  MoveL 2530 to (-12.23, -53.59, 110) mm, rotated rx 180 ry 0 rz 180 deg; joints [26.087, 43.16, 28.85, -152.762, 73.896, -188.126]
  Call Extruder(23965.750)
  MoveL 2531 to (0, -54.97, 110) mm, rotated rx 180 ry 0 rz -180 deg; joints [25.019, 44.364, 26.268, -153.678, 72.511, -188.456]
  Call Extruder(23973.266)
  MoveL 2532 to (8.41, -54.02, 110) mm, rotated rx -180 ry 0 rz 180 deg; joints [24.593, 45.312, 24.248, -153.968, 71.486, -188.816]
  Call Extruder(23976.680)
  MoveL 2533 to (12.23, -53.59, 110) mm, rotated rx -180 ry 0 rz -180 deg; joints [24.406, 45.751, 23.319, -154.09, 71.016, -188.98]
  Call Extruder(23987.610)
  MoveL 2534 to (23.85, -49.53, 110) mm, rotated rx 180 ry 0 rz 180 deg; joints [24.239, 47.254, 20.153, -154.003, 69.493, -189.695]
  Call Extruder(23998.541)
  MoveL 2535 to (34.27, -42.98, 110) mm, rotated rx -180 ry 0 rz 180 deg; joints [24.487, 48.8, 16.924, -153.451, 68.027, -190.589]
  Call Extruder(24009.471)
  MoveL 2536 to (42.98, -34.27, 110) mm, rotated rx -180 ry 0 rz -180 deg; joints [25.101, 50.315, 13.782, -152.49, 66.697, -191.641]
  Call Extruder(24020.401)
  MoveL 2537 to (49.52, -23.85, 110) mm, rotated rx 180 ry 0 rz 180 deg; joints [26.025, 51.725, 10.877, -151.191, 65.574, -192.812]
  Call Extruder(24031.331)
  MoveL 2538 to (53.59, -12.23, 110) mm, rotated rx 180 ry 0 rz -180 deg; joints [27.2, 52.961, 8.346, -149.634, 64.721, -194.047]
  Call Extruder(24042.261)
  MoveL 2539 to (54.97, 0, 110) mm, rotated rx 180 ry 0 rz 180 deg; joints [28.57, 53.956, 6.315, -147.909, 64.182, -195.275]
  Call Extruder(24053.192)
  MoveL 2540 to (53.59, 12.23, 110) mm, rotated rx 180 ry 0 rz -180 deg; joints [30.077, 54.657, 4.889, -146.106, 63.985, -196.418]
  Call Extruder(24064.122)
  MoveL 2541 to (49.52, 23.85, 110) mm, rotated rx -180 ry 0 rz -180 deg; joints [31.665, 55.023, 4.145, -144.311, 64.137, -197.398]
  Call Extruder(24075.052)
  MoveL 2542 to (42.98, 34.27, 110) mm, rotated rx -180 ry 0 rz -180 deg; joints [33.282, 55.034, 4.123, -142.6, 64.622, -198.143]
  Call Extruder(24085.982)
  MoveL 2543 to (34.27, 42.98, 110) mm, rotated rx 180 ry 0 rz -180 deg; joints [34.874, 54.688, 4.826, -141.036, 65.404, -198.604]
  Call Extruder(24096.912)
  MoveL 2544 to (23.85, 49.53, 110) mm, rotated rx -180 ry 0 rz -180 deg; joints [36.387, 54.006, 6.213, -139.667, 66.431, -198.752]
  Call Extruder(24107.843)
  MoveL 2545 to (12.23, 53.59, 110) mm, rotated rx 180 ry 0 rz 180 deg; joints [37.766, 53.026, 8.211, -138.531, 67.643, -198.581]
  Call Extruder(24118.773)
  MoveL 2546 to (0, 54.97, 110) mm, rotated rx 180 ry 0 rz -180 deg; joints [38.954, 51.803, 10.716, -137.657, 68.971, -198.108]
  Call Extruder(24129.703)
  MoveL 2547 to (-12.23, 53.59, 110) mm, rotated rx 180 ry 0 rz 180 deg; joints [39.895, 50.401, 13.604, -137.075, 70.35, -197.367]
  Call Extruder(24140.633)
  MoveL 2548 to (-23.85, 49.52, 110) mm, rotated rx 180 ry 0 rz 180 deg; joints [40.528, 48.89, 16.735, -136.814, 71.718, -196.406]
  Call Extruder(24151.563)
  MoveL 2549 to (-34.27, 42.98, 110) mm, rotated rx 180 ry 0 rz 180 deg; joints [40.799, 47.344, 19.964, -136.906, 73.02, -195.282]
  Call Extruder(24162.494)
  MoveL 2550 to (-42.98, 34.27, 110) mm, rotated rx 180 ry 0 rz 180 deg; joints [40.659, 45.837, 23.137, -137.381, 74.206, -194.06]
  Call Extruder(24173.424)
  MoveL 2551 to (-49.53, 23.85, 110) mm, rotated rx 180 ry 0 rz 180 deg; joints [40.072, 44.441, 26.103, -138.261, 75.233, -192.812]
  Call Extruder(24184.354)
  MoveL 2552 to (-53.59, 12.23, 110) mm, rotated rx 180 ry 0 rz 180 deg; joints [39.031, 43.225, 28.711, -139.546, 76.062, -191.607]
  Call Extruder(24195.284)
  MoveL 2553 to (-54.97, 0, 110) mm, rotated rx 180 ry 0 rz -180 deg; joints [37.56, 42.249, 30.821, -141.207, 76.654, -190.512]
  Call Extruder(24200.810)
  MoveL 2554 to (-54.27, -6.18, 110) mm, rotated rx 180 ry 0 rz 180 deg; joints [36.644, 41.897, 31.587, -142.193, 76.815, -190.036]
  Set speed (130.0 mm/s)
  MoveL 2555 to (-49.9, -9.51, 110) mm, rotated rx 180 ry 0 rz -180 deg; joints [35.741, 42.07, 31.21, -143.077, 76.496, -189.952]
  MoveL 2556 to (2.97, -12.99, 110) mm, rotated rx 180 ry 0 rz 180 deg; joints [30.614, 47.041, 20.6, -147.387, 70.89, -191.831]
  Call Extruder(24205.473)
  Set speed (80.0 mm/s)
  MoveL 2557 to (5.78, -12.01, 110) mm, rotated rx 180 ry 0 rz 180 deg; joints [30.526, 47.405, 19.836, -147.403, 70.534, -192.029]
  Call Extruder(24210.137)
  MoveL 2558 to (8.31, -10.42, 110) mm, rotated rx 180 ry 0 rz 180 deg; joints [30.538, 47.78, 19.051, -147.312, 70.192, -192.268]
  Call Extruder(24214.801)
  MoveL 2559 to (10.42, -8.31, 110) mm, rotated rx 180 ry 0 rz 180 deg; joints [30.649, 48.146, 18.287, -147.118, 69.881, -192.537]
  Call Extruder(24219.465)
  MoveL 2560 to (12.01, -5.78, 110) mm, rotated rx 180 ry 0 rz 180 deg; joints [30.85, 48.485, 17.579, -146.835, 69.616, -192.823]
  Call Extruder(24224.128)
  MoveL 2561 to (12.99, -2.97, 110) mm, rotated rx 180 ry 0 rz -180 deg; joints [31.131, 48.78, 16.965, -146.478, 69.412, -193.113]
  Call Extruder(24228.792)
  MoveL 2562 to (13.33, 0, 110) mm, rotated rx -180 ry 0 rz -180 deg; joints [31.476, 49.016, 16.474, -146.065, 69.279, -193.391]
  Call Extruder(24233.456)
  MoveL 2563 to (12.99, 2.97, 110) mm, rotated rx 180 ry 0 rz 180 deg; joints [31.869, 49.181, 16.131, -145.619, 69.224, -193.643]
  Call Extruder(24238.120)
  MoveL 2564 to (12.01, 5.78, 110) mm, rotated rx 180 ry 0 rz -180 deg; joints [32.292, 49.267, 15.952, -145.159, 69.248, -193.854]
  Call Extruder(24242.783)
  MoveL 2565 to (10.42, 8.31, 110) mm, rotated rx -180 ry 0 rz 180 deg; joints [32.725, 49.27, 15.947, -144.709, 69.35, -194.015]
  Call Extruder(24247.448)
  MoveL 2566 to (8.31, 10.42, 110) mm, rotated rx -180 ry 0 rz -180 deg; joints [33.149, 49.188, 16.116, -144.289, 69.524, -194.115]
  Call Extruder(24252.111)
  MoveL 2567 to (5.78, 12.01, 110) mm, rotated rx -180 ry 0 rz -180 deg; joints [33.544, 49.027, 16.45, -143.918, 69.761, -194.149]
  Call Extruder(24256.775)
  MoveL 2568 to (2.97, 13, 110) mm, rotated rx -180 ry 0 rz -180 deg; joints [33.893, 48.795, 16.933, -143.612, 70.049, -194.115]
  Call Extruder(24261.439)
  MoveL 2569 to (0, 13.33, 110) mm, rotated rx -180 ry 0 rz 180 deg; joints [34.177, 48.503, 17.54, -143.386, 70.372, -194.014]
  Call Extruder(24266.103)
  MoveL 2570 to (-2.97, 13, 110) mm, rotated rx 180 ry 0 rz 180 deg; joints [34.384, 48.167, 18.243, -143.251, 70.715, -193.854]
  Call Extruder(24270.766)
  MoveL 2571 to (-5.78, 12.01, 110) mm, rotated rx 180 ry 0 rz 180 deg; joints [34.5, 47.802, 19.005, -143.214, 71.061, -193.641]
  Call Extruder(24275.430)
  MoveL 2572 to (-8.31, 10.42, 110) mm, rotated rx 180 ry 0 rz -180 deg; joints [34.518, 47.427, 19.79, -143.279, 71.393, -193.388]
  Call Extruder(24280.094)
  MoveL 2573 to (-10.42, 8.31, 110) mm, rotated rx 180 ry 0 rz -180 deg; joints [34.436, 47.061, 20.556, -143.443, 71.696, -193.109]
  Call Extruder(24284.758)
  MoveL 2574 to (-12.01, 5.78, 110) mm, rotated rx 180 ry 0 rz -180 deg; joints [34.254, 46.723, 21.268, -143.702, 71.956, -192.818]
  Call Extruder(24289.421)
  MoveL 2575 to (-12.99, 2.97, 110) mm, rotated rx -180 ry 0 rz -180 deg; joints [33.981, 46.429, 21.887, -144.044, 72.158, -192.53]
  Call Extruder(24294.085)
  MoveL 2576 to (-13.33, 0, 110) mm, rotated rx 180 ry 0 rz -180 deg; joints [33.63, 46.194, 22.383, -144.454, 72.295, -192.26]
  Call Extruder(24298.749)
  MoveL 2577 to (-13, -2.97, 110) mm, rotated rx 180 ry 0 rz 180 deg; joints [33.218, 46.029, 22.731, -144.91, 72.357, -192.02]
  Call Extruder(24303.413)
  MoveL 2578 to (-12.01, -5.78, 110) mm, rotated rx -180 ry 0 rz -180 deg; joints [32.767, 45.943, 22.912, -145.39, 72.343, -191.823]
  Call Extruder(24308.076)
  MoveL 2579 to (-10.42, -8.31, 110) mm, rotated rx -180 ry 0 rz -180 deg; joints [32.302, 45.941, 22.917, -145.868, 72.25, -191.676]
  Call Extruder(24312.741)
  MoveL 2580 to (-8.31, -10.42, 110) mm, rotated rx 180 ry 0 rz 180 deg; joints [31.85, 46.022, 22.746, -146.317, 72.084, -191.586]
  Call Extruder(24317.404)
  MoveL 2581 to (-5.78, -12.01, 110) mm, rotated rx 180 ry 0 rz -180 deg; joints [31.435, 46.182, 22.408, -146.713, 71.853, -191.557]
  Call Extruder(24322.068)
  MoveL 2582 to (-2.97, -12.99, 110) mm, rotated rx 180 ry 0 rz -180 deg; joints [31.079, 46.413, 21.92, -147.034, 71.566, -191.59]
  Call Extruder(24326.732)
  MoveL 2583 to (0, -13.33, 110) mm, rotated rx 180 ry 0 rz 180 deg; joints [30.801, 46.704, 21.307, -147.262, 71.24, -191.682]
  Call Extruder(24331.396)
  MoveL 2584 to (2.97, -12.99, 110) mm, rotated rx 180 ry 0 rz 180 deg; joints [30.614, 47.041, 20.6, -147.387, 70.89, -191.831]
  Set speed (130.0 mm/s)
  MoveL 2585 to (2.97, -12.99, 115) mm, rotated rx 180 ry 0 rz 180 deg; joints [30.614, 46.171, 20.829, -147.266, 70.35, -192.198]
  MoveL 2586 to (-26.25, -4.54, 115) mm, rotated rx 180 ry 0 rz 180 deg; joints [34.172, 43.696, 25.979, -144.096, 73.299, -191.753]
  Call Extruder(24333.628)
  Set speed (60.0 mm/s)
  MoveL 2587 to (-26.09, -5.96, 115) mm, rotated rx 180 ry 0 rz -180 deg; joints [33.969, 43.617, 26.145, -144.319, 73.328, -191.64]
  Call Extruder(24342.993)
  MoveL 2588 to (-24.12, -11.61, 115) mm, rotated rx -180 ry 0 rz 180 deg; joints [33.033, 43.441, 26.513, -145.31, 73.3, -191.25]
  Call Extruder(24352.358)
  MoveL 2589 to (-20.93, -16.69, 115) mm, rotated rx -180 ry 0 rz -180 deg; joints [32.066, 43.436, 26.524, -146.303, 73.118, -190.96]
  Call Extruder(24361.723)
  MoveL 2590 to (-16.69, -20.93, 115) mm, rotated rx 180 ry 0 rz 180 deg; joints [31.126, 43.602, 26.176, -147.237, 72.789, -190.781]
  Call Extruder(24371.088)
  MoveL 2591 to (-11.61, -24.11, 115) mm, rotated rx 180 ry 0 rz -180 deg; joints [30.272, 43.93, 25.489, -148.057, 72.326, -190.719]
  Call Extruder(24380.453)
  MoveL 2592 to (-5.96, -26.09, 115) mm, rotated rx 180 ry 0 rz -180 deg; joints [29.552, 44.403, 24.5, -148.713, 71.753, -190.773]
  Call Extruder(24389.818)
  MoveL 2593 to (0, -26.77, 115) mm, rotated rx 180 ry 0 rz -180 deg; joints [29.003, 44.998, 23.261, -149.17, 71.098, -190.943]
  Call Extruder(24399.183)
  MoveL 2594 to (5.96, -26.09, 115) mm, rotated rx 180 ry 0 rz 180 deg; joints [28.65, 45.685, 21.836, -149.405, 70.395, -191.222]
  Call Extruder(24408.548)
  MoveL 2595 to (11.61, -24.12, 115) mm, rotated rx -180 ry 0 rz -180 deg; joints [28.503, 46.429, 20.297, -149.412, 69.681, -191.599]
  Call Extruder(24417.913)
  MoveL 2596 to (16.69, -20.93, 115) mm, rotated rx 180 ry 0 rz 180 deg; joints [28.559, 47.193, 18.722, -149.196, 68.995, -192.063]
  Call Extruder(24427.278)
  MoveL 2597 to (20.93, -16.69, 115) mm, rotated rx 180 ry 0 rz -180 deg; joints [28.808, 47.939, 17.188, -148.777, 68.374, -192.593]
  Call Extruder(24436.643)
  MoveL 2598 to (24.12, -11.61, 115) mm, rotated rx 180 ry 0 rz 180 deg; joints [29.229, 48.631, 15.771, -148.183, 67.849, -193.167]
  Call Extruder(24446.008)
  MoveL 2599 to (26.09, -5.96, 115) mm, rotated rx 180 ry 0 rz -180 deg; joints [29.796, 49.233, 14.54, -147.448, 67.449, -193.756]
  Call Extruder(24455.373)
  MoveL 2600 to (26.77, 0, 115) mm, rotated rx -180 ry 0 rz 180 deg; joints [30.482, 49.715, 13.556, -146.614, 67.194, -194.33]
  Call Extruder(24464.738)
  MoveL 2601 to (26.09, 5.96, 115) mm, rotated rx 180 ry 0 rz -180 deg; joints [31.252, 50.053, 12.867, -145.722, 67.097, -194.856]
  Call Extruder(24474.103)
  MoveL 2602 to (24.12, 11.61, 115) mm, rotated rx 180 ry 0 rz -180 deg; joints [32.076, 50.229, 12.509, -144.815, 67.162, -195.304]
  Call Extruder(24483.468)
  MoveL 2603 to (20.93, 16.69, 115) mm, rotated rx 180 ry 0 rz -180 deg; joints [32.917, 50.234, 12.499, -143.935, 67.382, -195.647]
  Call Extruder(24492.833)
  MoveL 2604 to (16.69, 20.93, 115) mm, rotated rx 180 ry 0 rz -180 deg; joints [33.742, 50.068, 12.837, -143.118, 67.744, -195.864]
  Call Extruder(24502.198)
  MoveL 2605 to (11.61, 24.12, 115) mm, rotated rx 180 ry 0 rz -180 deg; joints [34.517, 49.739, 13.507, -142.397, 68.228, -195.943]
  Call Extruder(24511.563)
  MoveL 2606 to (5.96, 26.09, 115) mm, rotated rx -180 ry 0 rz -180 deg; joints [35.208, 49.265, 14.475, -141.802, 68.807, -195.879]
  Call Extruder(24520.928)
  MoveL 2607 to (0, 26.77, 115) mm, rotated rx 180 ry 0 rz 180 deg; joints [35.784, 48.669, 15.692, -141.357, 69.451, -195.676]
  Call Extruder(24530.293)
  MoveL 2608 to (-5.96, 26.09, 115) mm, rotated rx 180 ry 0 rz -180 deg; joints [36.214, 47.982, 17.101, -141.082, 70.128, -195.348]
  Call Extruder(24539.658)
  MoveL 2609 to (-11.61, 24.12, 115) mm, rotated rx 180 ry 0 rz -180 deg; joints [36.473, 47.238, 18.63, -140.991, 70.806, -194.913]
  Call Extruder(24549.023)
  MoveL 2610 to (-16.69, 20.93, 115) mm, rotated rx 180 ry 0 rz -180 deg; joints [36.542, 46.474, 20.205, -141.096, 71.454, -194.397]
  Call Extruder(24558.388)
  MoveL 2611 to (-20.93, 16.69, 115) mm, rotated rx 180 ry 0 rz 180 deg; joints [36.407, 45.728, 21.747, -141.398, 72.042, -193.828]
  Call Extruder(24567.753)
  MoveL 2612 to (-24.12, 11.61, 115) mm, rotated rx 180 ry 0 rz -180 deg; joints [36.065, 45.037, 23.182, -141.894, 72.545, -193.238]
  Call Extruder(24577.118)
  MoveL 2613 to (-26.09, 5.96, 115) mm, rotated rx 180 ry 0 rz 180 deg; joints [35.528, 44.435, 24.434, -142.566, 72.939, -192.658]
  Call Extruder(24586.483)
  MoveL 2614 to (-26.77, 0, 115) mm, rotated rx 180 ry 0 rz 180 deg; joints [34.817, 43.954, 25.439, -143.388, 73.205, -192.117]
  Call Extruder(24591.271)
  MoveL 2615 to (-26.42, -3.05, 115) mm, rotated rx 180 ry 0 rz 180 deg; joints [34.385, 43.78, 25.803, -143.863, 73.268, -191.872]
  Set speed (130.0 mm/s)
  MoveL 2616 to (-41.86, -6.29, 115) mm, rotated rx -180 ry 0 rz 180 deg; joints [35.393, 42.068, 29.404, -143.155, 74.986, -190.985]
  Call Extruder(24596.269)
  Set speed (60.0 mm/s)
  MoveL 2617 to (-41.5, -9.47, 115) mm, rotated rx 180 ry 0 rz -180 deg; joints [34.924, 41.89, 29.78, -143.664, 75.057, -190.74]
  Call Extruder(24611.165)
  MoveL 2618 to (-38.36, -18.47, 115) mm, rotated rx 180 ry 0 rz 180 deg; joints [33.373, 41.609, 30.376, -145.291, 75.032, -190.143]
  Call Extruder(24626.061)
  MoveL 2619 to (-33.29, -26.54, 115) mm, rotated rx -180 ry 0 rz 180 deg; joints [31.763, 41.6, 30.393, -146.935, 74.762, -189.709]
  Call Extruder(24640.957)
  MoveL 2620 to (-26.54, -33.29, 115) mm, rotated rx -180 ry 0 rz 180 deg; joints [30.206, 41.866, 29.831, -148.484, 74.252, -189.449]
  Call Extruder(24655.852)
  MoveL 2621 to (-18.47, -38.36, 115) mm, rotated rx 180 ry 0 rz -180 deg; joints [28.808, 42.391, 28.721, -149.834, 73.522, -189.362]
  Call Extruder(24670.748)
  MoveL 2622 to (-9.47, -41.5, 115) mm, rotated rx 180 ry 0 rz 180 deg; joints [27.654, 43.148, 27.128, -150.897, 72.606, -189.448]
  Call Extruder(24685.644)
  MoveL 2623 to (0, -42.57, 115) mm, rotated rx 180 ry 0 rz -180 deg; joints [26.805, 44.097, 25.141, -151.616, 71.554, -189.702]
  Call Extruder(24697.356)
  MoveL 2624 to (7.45, -41.73, 115) mm, rotated rx 180 ry 0 rz 180 deg; joints [26.398, 44.954, 23.354, -151.89, 70.665, -190.03]
  Call Extruder(24700.540)
  MoveL 2625 to (9.47, -41.5, 115) mm, rotated rx 180 ry 0 rz 180 deg; joints [26.29, 45.19, 22.863, -151.96, 70.422, -190.119]
  Call Extruder(24715.435)
  MoveL 2626 to (18.47, -38.36, 115) mm, rotated rx 180 ry 0 rz -180 deg; joints [26.114, 46.373, 20.412, -151.925, 69.271, -190.691]
  Call Extruder(24730.331)
  MoveL 2627 to (26.54, -33.28, 115) mm, rotated rx 180 ry 0 rz 180 deg; joints [26.262, 47.588, 17.908, -151.532, 68.165, -191.402]
  Call Extruder(24745.227)
  MoveL 2628 to (33.28, -26.54, 115) mm, rotated rx 180 ry 0 rz -180 deg; joints [26.703, 48.777, 15.472, -150.817, 67.162, -192.23]
  Call Extruder(24760.123)
  MoveL 2629 to (38.36, -18.47, 115) mm, rotated rx 180 ry 0 rz 180 deg; joints [27.4, 49.879, 13.221, -149.833, 66.317, -193.141]
  Call Extruder(24775.019)
  MoveL 2630 to (41.51, -9.47, 115) mm, rotated rx 180 ry 0 rz 180 deg; joints [28.309, 50.841, 11.265, -148.64, 65.677, -194.091]
  Call Extruder(24789.914)
  MoveL 2631 to (42.57, 0, 115) mm, rotated rx 180 ry 0 rz 180 deg; joints [29.382, 51.614, 9.698, -147.305, 65.273, -195.029]
  Call Extruder(24804.810)
  MoveL 2632 to (41.5, 9.47, 115) mm, rotated rx 180 ry 0 rz 180 deg; joints [30.575, 52.156, 8.601, -145.898, 65.128, -195.896]
  Call Extruder(24819.706)
  MoveL 2633 to (38.36, 18.47, 115) mm, rotated rx -180 ry 0 rz -180 deg; joints [31.839, 52.439, 8.028, -144.485, 65.244, -196.639]
  Call Extruder(24834.602)
  MoveL 2634 to (33.28, 26.54, 115) mm, rotated rx -180 ry 0 rz 180 deg; joints [33.128, 52.447, 8.012, -143.127, 65.613, -197.208]
  Call Extruder(24849.498)
  MoveL 2635 to (26.54, 33.29, 115) mm, rotated rx 180 ry 0 rz 180 deg; joints [34.394, 52.18, 8.552, -141.877, 66.208, -197.567]
  Call Extruder(24864.394)
  MoveL 2636 to (18.47, 38.36, 115) mm, rotated rx -180 ry 0 rz 180 deg; joints [35.592, 51.653, 9.62, -140.779, 66.992, -197.693]
  Call Extruder(24879.289)
  MoveL 2637 to (9.47, 41.51, 115) mm, rotated rx -180 ry 0 rz -180 deg; joints [36.675, 50.892, 11.161, -139.869, 67.922, -197.581]
  Call Extruder(24894.185)
  MoveL 2638 to (0, 42.57, 115) mm, rotated rx 180 ry 0 rz -180 deg; joints [37.594, 49.94, 13.097, -139.178, 68.945, -197.241]
  Call Extruder(24909.081)
  MoveL 2639 to (-9.47, 41.51, 115) mm, rotated rx 180 ry 0 rz 180 deg; joints [38.304, 48.844, 15.334, -138.733, 70.013, -196.696]
  Call Extruder(24923.977)
  MoveL 2640 to (-18.47, 38.36, 115) mm, rotated rx -180 ry 0 rz 180 deg; joints [38.762, 47.66, 17.762, -138.557, 71.075, -195.98]
  Call Extruder(24938.872)
  MoveL 2641 to (-26.54, 33.28, 115) mm, rotated rx -180 ry 0 rz -180 deg; joints [38.928, 46.444, 20.265, -138.672, 72.086, -195.136]
  Call Extruder(24953.768)
  MoveL 2642 to (-33.29, 26.54, 115) mm, rotated rx 180 ry 0 rz -180 deg; joints [38.772, 45.258, 22.723, -139.094, 73.004, -194.212]
  Call Extruder(24968.664)
  MoveL 2643 to (-38.36, 18.47, 115) mm, rotated rx 180 ry 0 rz 180 deg; joints [38.277, 44.157, 25.013, -139.826, 73.791, -193.261]
  Call Extruder(24983.560)
  MoveL 2644 to (-41.5, 9.47, 115) mm, rotated rx -180 ry 0 rz 180 deg; joints [37.447, 43.199, 27.021, -140.859, 74.415, -192.334]
  Call Extruder(24998.456)
  MoveL 2645 to (-42.57, 0, 115) mm, rotated rx 180 ry 0 rz -180 deg; joints [36.31, 42.429, 28.64, -142.158, 74.845, -191.48]
  Call Extruder(25006.010)
  MoveL 2646 to (-42.03, -4.8, 115) mm, rotated rx 180 ry 0 rz 180 deg; joints [35.612, 42.152, 29.225, -142.917, 74.953, -191.101]
  Set speed (130.0 mm/s)
  MoveL 2647 to (-54.1, -7.67, 115) mm, rotated rx 180 ry 0 rz -180 deg; joints [36.421, 40.842, 32.007, -142.326, 76.273, -190.383]
  Call Extruder(25010.083)
  Set speed (30.0 mm/s)
  MoveL 2648 to (-53.59, -12.23, 115) mm, rotated rx -180 ry 0 rz -180 deg; joints [35.732, 40.586, 32.552, -143.067, 76.381, -190.038]
  Call Extruder(25021.013)
  MoveL 2649 to (-49.53, -23.85, 115) mm, rotated rx 180 ry 0 rz 180 deg; joints [33.663, 40.22, 33.335, -145.224, 76.372, -189.292]
  Call Extruder(25031.943)
  MoveL 2650 to (-42.98, -34.27, 115) mm, rotated rx 180 ry 0 rz -180 deg; joints [31.506, 40.21, 33.357, -147.42, 76.043, -188.762]
  Call Extruder(25042.873)
  MoveL 2651 to (-34.27, -42.98, 115) mm, rotated rx 180 ry 0 rz -180 deg; joints [29.427, 40.555, 32.618, -149.488, 75.397, -188.451]
  Call Extruder(25053.803)
  MoveL 2652 to (-23.85, -49.52, 115) mm, rotated rx -180 ry 0 rz -180 deg; joints [27.581, 41.237, 31.165, -151.277, 74.456, -188.354]
  Call Extruder(25064.734)
  MoveL 2653 to (-12.23, -53.59, 115) mm, rotated rx 180 ry 0 rz 180 deg; joints [26.087, 42.218, 29.086, -152.666, 73.268, -188.464]
  Call Extruder(25075.664)
  MoveL 2654 to (0, -54.97, 115) mm, rotated rx 180 ry 0 rz 180 deg; joints [25.019, 43.447, 26.501, -153.581, 71.898, -188.775]
  Call Extruder(25083.552)
  MoveL 2655 to (8.83, -53.97, 115) mm, rotated rx 180 ry 0 rz 180 deg; joints [24.572, 44.462, 24.378, -153.881, 70.835, -189.144]
  Call Extruder(25086.594)
  MoveL 2656 to (12.23, -53.59, 115) mm, rotated rx 180 ry 0 rz 180 deg; joints [24.406, 44.86, 23.549, -153.989, 70.422, -189.287]
  Call Extruder(25097.524)
  MoveL 2657 to (23.85, -49.52, 115) mm, rotated rx 180 ry 0 rz -180 deg; joints [24.239, 46.388, 20.382, -153.897, 68.921, -189.994]
  Call Extruder(25108.454)
  MoveL 2658 to (34.27, -42.98, 115) mm, rotated rx 180 ry 0 rz 180 deg; joints [24.487, 47.957, 17.151, -153.339, 67.477, -190.887]
  Call Extruder(25119.384)
  MoveL 2659 to (42.98, -34.27, 115) mm, rotated rx 180 ry 0 rz 180 deg; joints [25.101, 49.493, 14.009, -152.37, 66.169, -191.942]
  Call Extruder(25130.315)
  MoveL 2660 to (49.52, -23.85, 115) mm, rotated rx 180 ry 0 rz -180 deg; joints [26.025, 50.921, 11.103, -151.063, 65.068, -193.119]
  Call Extruder(25141.245)
  MoveL 2661 to (53.59, -12.23, 115) mm, rotated rx 180 ry 0 rz 180 deg; joints [27.2, 52.17, 8.573, -149.498, 64.235, -194.363]
  Call Extruder(25152.175)
  MoveL 2662 to (54.97, 0, 115) mm, rotated rx 180 ry 0 rz -180 deg; joints [28.57, 53.175, 6.543, -147.765, 63.714, -195.603]
  Call Extruder(25163.105)
  MoveL 2663 to (53.59, 12.23, 115) mm, rotated rx 180 ry 0 rz 180 deg; joints [30.077, 53.883, 5.118, -145.956, 63.533, -196.758]
  Call Extruder(25174.035)
  MoveL 2664 to (49.52, 23.85, 115) mm, rotated rx 180 ry 0 rz 180 deg; joints [31.665, 54.253, 4.374, -144.156, 63.698, -197.75]
  Call Extruder(25184.966)
  MoveL 2665 to (42.98, 34.27, 115) mm, rotated rx 180 ry 0 rz -180 deg; joints [33.282, 54.264, 4.352, -142.442, 64.192, -198.508]
  Call Extruder(25195.896)
  MoveL 2666 to (34.27, 42.98, 115) mm, rotated rx 180 ry 0 rz 180 deg; joints [34.874, 53.914, 5.054, -140.877, 64.981, -198.982]
  Call Extruder(25206.826)
  MoveL 2667 to (23.85, 49.53, 115) mm, rotated rx 180 ry 0 rz -180 deg; joints [36.387, 53.226, 6.441, -139.51, 66.011, -199.143]
  Call Extruder(25217.756)
  MoveL 2668 to (12.23, 53.59, 115) mm, rotated rx 180 ry 0 rz -180 deg; joints [37.766, 52.236, 8.438, -138.376, 67.221, -198.985]
  Call Extruder(25228.687)
  MoveL 2669 to (0, 54.97, 115) mm, rotated rx 180 ry 0 rz -180 deg; joints [38.954, 51, 10.943, -137.506, 68.545, -198.526]
  Call Extruder(25239.617)
  MoveL 2670 to (-12.23, 53.59, 115) mm, rotated rx 180 ry 0 rz -180 deg; joints [39.895, 49.581, 13.83, -136.929, 69.916, -197.798]
  Call Extruder(25250.547)
  MoveL 2671 to (-23.85, 49.52, 115) mm, rotated rx 180 ry 0 rz -180 deg; joints [40.528, 48.049, 16.962, -136.673, 71.271, -196.85]
  Call Extruder(25261.477)
  MoveL 2672 to (-34.27, 42.98, 115) mm, rotated rx 180 ry 0 rz 180 deg; joints [40.799, 46.48, 20.192, -136.772, 72.556, -195.737]
  Call Extruder(25272.407)
  MoveL 2673 to (-42.98, 34.27, 115) mm, rotated rx 180 ry 0 rz 180 deg; joints [40.659, 44.947, 23.367, -137.253, 73.721, -194.525]
  Call Extruder(25283.338)
  MoveL 2674 to (-49.53, 23.85, 115) mm, rotated rx -180 ry 0 rz 180 deg; joints [40.072, 43.525, 26.336, -138.139, 74.724, -193.283]
  Call Extruder(25294.268)
  MoveL 2675 to (-53.59, 12.23, 115) mm, rotated rx -180 ry 0 rz -180 deg; joints [39.031, 42.284, 28.946, -139.43, 75.526, -192.079]
  Call Extruder(25305.198)
  MoveL 2676 to (-54.97, 0, 115) mm, rotated rx 180 ry 0 rz 180 deg; joints [37.56, 41.287, 31.059, -141.096, 76.089, -190.979]
  Call Extruder(25310.724)
  MoveL 2677 to (-54.27, -6.18, 115) mm, rotated rx 180 ry 0 rz 180 deg; joints [36.644, 40.927, 31.826, -142.085, 76.237, -190.498]
  Set speed (130.0 mm/s)
  MoveL 2678 to (-49.9, -9.51, 115) mm, rotated rx 180 ry 0 rz 180 deg; joints [35.741, 41.104, 31.448, -142.97, 75.915, -190.403]
  MoveL 2679 to (2.97, -12.99, 115) mm, rotated rx 180 ry 0 rz 180 deg; joints [30.614, 46.171, 20.829, -147.266, 70.35, -192.198]
  Call Extruder(25315.387)
  Set speed (80.0 mm/s)
  MoveL 2680 to (5.78, -12.01, 115) mm, rotated rx 180 ry 0 rz -180 deg; joints [30.526, 46.542, 20.064, -147.28, 70, -192.393]
  Call Extruder(25320.051)
  MoveL 2681 to (8.31, -10.42, 115) mm, rotated rx -180 ry 0 rz -180 deg; joints [30.538, 46.922, 19.279, -147.187, 69.662, -192.631]
  Call Extruder(25324.715)
  MoveL 2682 to (10.42, -8.31, 115) mm, rotated rx 180 ry 0 rz -180 deg; joints [30.649, 47.294, 18.514, -146.992, 69.357, -192.899]
  Call Extruder(25329.379)
  MoveL 2683 to (12.01, -5.78, 115) mm, rotated rx -180 ry 0 rz 180 deg; joints [30.85, 47.638, 17.807, -146.707, 69.098, -193.186]
  Call Extruder(25334.042)
  MoveL 2684 to (12.99, -2.97, 115) mm, rotated rx 180 ry 0 rz 180 deg; joints [31.131, 47.937, 17.192, -146.348, 68.899, -193.477]
  Call Extruder(25338.706)
  MoveL 2685 to (13.33, 0, 115) mm, rotated rx 180 ry 0 rz 180 deg; joints [31.476, 48.176, 16.701, -145.934, 68.772, -193.757]
  Call Extruder(25343.370)
  MoveL 2686 to (12.99, 2.97, 115) mm, rotated rx -180 ry 0 rz -180 deg; joints [31.869, 48.344, 16.358, -145.486, 68.721, -194.012]
  Call Extruder(25348.034)
  MoveL 2687 to (12.01, 5.78, 115) mm, rotated rx -180 ry 0 rz -180 deg; joints [32.292, 48.431, 16.179, -145.026, 68.749, -194.228]
  Call Extruder(25352.697)
  MoveL 2688 to (10.42, 8.31, 115) mm, rotated rx -180 ry 0 rz -180 deg; joints [32.725, 48.434, 16.174, -144.575, 68.854, -194.392]
  Call Extruder(25357.361)
  MoveL 2689 to (8.31, 10.42, 115) mm, rotated rx -180 ry 0 rz 180 deg; joints [33.149, 48.352, 16.342, -144.154, 69.03, -194.496]
  Call Extruder(25362.025)
  MoveL 2690 to (5.78, 12.01, 115) mm, rotated rx 180 ry 0 rz -180 deg; joints [33.544, 48.188, 16.677, -143.783, 69.267, -194.534]
  Call Extruder(25366.689)
  MoveL 2691 to (2.97, 13, 115) mm, rotated rx 180 ry 0 rz 180 deg; joints [33.893, 47.953, 17.16, -143.478, 69.554, -194.504]
  Call Extruder(25371.353)
  MoveL 2692 to (0, 13.33, 115) mm, rotated rx 180 ry 0 rz -180 deg; joints [34.177, 47.657, 17.768, -143.253, 69.875, -194.408]
  Call Extruder(25376.017)
  MoveL 2693 to (-2.97, 12.99, 115) mm, rotated rx 180 ry 0 rz 180 deg; joints [34.384, 47.315, 18.47, -143.119, 70.215, -194.25]
  Call Extruder(25380.680)
  MoveL 2694 to (-5.78, 12.01, 115) mm, rotated rx -180 ry 0 rz 180 deg; joints [34.5, 46.945, 19.233, -143.083, 70.557, -194.04]
  Call Extruder(25385.344)
  MoveL 2695 to (-8.31, 10.42, 115) mm, rotated rx 180 ry 0 rz 180 deg; joints [34.518, 46.564, 20.018, -143.149, 70.885, -193.79]
  Call Extruder(25390.008)
  MoveL 2696 to (-10.42, 8.31, 115) mm, rotated rx -180 ry 0 rz 180 deg; joints [34.436, 46.193, 20.785, -143.315, 71.182, -193.512]
  Call Extruder(25394.672)
  MoveL 2697 to (-12.01, 5.78, 115) mm, rotated rx 180 ry 0 rz -180 deg; joints [34.254, 45.849, 21.497, -143.575, 71.436, -193.221]
  Call Extruder(25399.335)
  MoveL 2698 to (-13, 2.97, 115) mm, rotated rx 180 ry 0 rz -180 deg; joints [33.981, 45.55, 22.116, -143.919, 71.633, -192.932]
  Call Extruder(25403.999)
  MoveL 2699 to (-13.33, 0, 115) mm, rotated rx 180 ry 0 rz 180 deg; joints [33.63, 45.31, 22.613, -144.33, 71.763, -192.66]
  Call Extruder(25408.663)
  MoveL 2700 to (-13, -2.97, 115) mm, rotated rx 180 ry 0 rz -180 deg; joints [33.218, 45.143, 22.961, -144.788, 71.821, -192.417]
  Call Extruder(25413.327)
  MoveL 2701 to (-12.01, -5.78, 115) mm, rotated rx 180 ry 0 rz 180 deg; joints [32.767, 45.056, 23.142, -145.269, 71.802, -192.216]
  Call Extruder(25417.990)
  MoveL 2702 to (-10.42, -8.31, 115) mm, rotated rx 180 ry 0 rz -180 deg; joints [32.302, 45.053, 23.147, -145.748, 71.706, -192.065]
  Call Extruder(25422.654)
  MoveL 2703 to (-8.31, -10.42, 115) mm, rotated rx 180 ry 0 rz 180 deg; joints [31.85, 45.135, 22.976, -146.197, 71.539, -191.97]
  Call Extruder(25427.318)
  MoveL 2704 to (-5.78, -12.01, 115) mm, rotated rx 180 ry 0 rz -180 deg; joints [31.435, 45.298, 22.638, -146.593, 71.306, -191.936]
  Call Extruder(25431.982)
  MoveL 2705 to (-2.97, -12.99, 115) mm, rotated rx 180 ry 0 rz -180 deg; joints [31.079, 45.534, 22.149, -146.914, 71.021, -191.964]
  Call Extruder(25436.646)
  MoveL 2706 to (0, -13.33, 115) mm, rotated rx -180 ry 0 rz 180 deg; joints [30.801, 45.83, 21.536, -147.142, 70.697, -192.052]
  Call Extruder(25441.310)
  MoveL 2707 to (2.97, -12.99, 115) mm, rotated rx 180 ry 0 rz 180 deg; joints [30.614, 46.171, 20.829, -147.266, 70.35, -192.198]
  Set speed (130.0 mm/s)
  MoveL 2708 to (2.97, -12.99, 120) mm, rotated rx -180 ry 0 rz 180 deg; joints [30.614, 45.309, 21.04, -147.138, 69.803, -192.573]
  MoveL 2709 to (-26.25, -4.54, 120) mm, rotated rx -180 ry 0 rz 180 deg; joints [34.172, 42.79, 26.194, -143.972, 72.739, -192.177]
  Call Extruder(25443.542)
  Set speed (60.0 mm/s)
  MoveL 2710 to (-26.09, -5.96, 120) mm, rotated rx 180 ry 0 rz 180 deg; joints [33.969, 42.709, 26.36, -144.196, 72.766, -192.063]
  Call Extruder(25452.907)
  MoveL 2711 to (-24.12, -11.61, 120) mm, rotated rx 180 ry 0 rz 180 deg; joints [33.033, 42.53, 26.728, -145.189, 72.728, -191.664]
  Call Extruder(25462.272)
  MoveL 2712 to (-20.93, -16.69, 120) mm, rotated rx 180 ry 0 rz -180 deg; joints [32.066, 42.525, 26.739, -146.184, 72.539, -191.364]
  Call Extruder(25471.637)
  MoveL 2713 to (-16.69, -20.93, 120) mm, rotated rx 180 ry 0 rz -180 deg; joints [31.126, 42.694, 26.391, -147.119, 72.207, -191.175]
  Call Extruder(25481.002)
  MoveL 2714 to (-11.61, -24.11, 120) mm, rotated rx 180 ry 0 rz 180 deg; joints [30.272, 43.028, 25.704, -147.939, 71.744, -191.101]
  Call Extruder(25490.367)
  MoveL 2715 to (-5.96, -26.09, 120) mm, rotated rx 180 ry 0 rz -180 deg; joints [29.552, 43.511, 24.714, -148.595, 71.173, -191.146]
  Call Extruder(25499.732)
  MoveL 2716 to (0, -26.77, 120) mm, rotated rx -180 ry 0 rz -180 deg; joints [29.003, 44.116, 23.474, -149.05, 70.523, -191.307]
  Call Extruder(25509.097)
  MoveL 2717 to (5.96, -26.09, 120) mm, rotated rx -180 ry 0 rz 180 deg; joints [28.65, 44.815, 22.047, -149.284, 69.828, -191.579]
  Call Extruder(25518.462)
  MoveL 2718 to (11.61, -24.12, 120) mm, rotated rx -180 ry 0 rz -180 deg; joints [28.503, 45.57, 20.508, -149.288, 69.125, -191.952]
  Call Extruder(25527.827)
  MoveL 2719 to (16.69, -20.93, 120) mm, rotated rx 180 ry 0 rz 180 deg; joints [28.559, 46.346, 18.932, -149.069, 68.449, -192.413]
  Call Extruder(25537.192)
  MoveL 2720 to (20.93, -16.69, 120) mm, rotated rx -180 ry 0 rz -180 deg; joints [28.808, 47.103, 17.398, -148.647, 67.839, -192.943]
  Call Extruder(25546.557)
  MoveL 2721 to (24.12, -11.61, 120) mm, rotated rx -180 ry 0 rz 180 deg; joints [29.229, 47.805, 15.98, -148.049, 67.325, -193.519]
  Call Extruder(25555.922)
  MoveL 2722 to (26.09, -5.96, 120) mm, rotated rx 180 ry 0 rz 180 deg; joints [29.796, 48.415, 14.749, -147.31, 66.936, -194.112]
  Call Extruder(25565.287)
  MoveL 2723 to (26.77, 0, 120) mm, rotated rx 180 ry 0 rz 180 deg; joints [30.482, 48.903, 13.765, -146.472, 66.691, -194.691]
  Call Extruder(25574.652)
  MoveL 2724 to (26.09, 5.96, 120) mm, rotated rx 180 ry 0 rz 180 deg; joints [31.252, 49.245, 13.077, -145.578, 66.603, -195.223]
  Call Extruder(25584.017)
  MoveL 2725 to (24.11, 11.61, 120) mm, rotated rx 180 ry 0 rz -180 deg; joints [32.076, 49.424, 12.718, -144.669, 66.675, -195.678]
  Call Extruder(25593.382)
  MoveL 2726 to (20.93, 16.69, 120) mm, rotated rx -180 ry 0 rz 180 deg; joints [32.917, 49.429, 12.708, -143.787, 66.9, -196.028]
  Call Extruder(25602.747)
  MoveL 2727 to (16.69, 20.93, 120) mm, rotated rx 180 ry 0 rz -180 deg; joints [33.742, 49.261, 13.046, -142.969, 67.266, -196.253]
  Call Extruder(25612.112)
  MoveL 2728 to (11.61, 24.12, 120) mm, rotated rx 180 ry 0 rz -180 deg; joints [34.517, 48.928, 13.716, -142.249, 67.751, -196.34]
  Call Extruder(25621.476)
  MoveL 2729 to (5.96, 26.09, 120) mm, rotated rx 180 ry 0 rz -180 deg; joints [35.208, 48.447, 14.684, -141.655, 68.329, -196.284]
  Call Extruder(25630.842)
  MoveL 2730 to (0, 26.77, 120) mm, rotated rx -180 ry 0 rz -180 deg; joints [35.784, 47.843, 15.902, -141.211, 68.97, -196.088]
  Call Extruder(25640.207)
  MoveL 2731 to (-5.96, 26.09, 120) mm, rotated rx 180 ry 0 rz -180 deg; joints [36.214, 47.147, 17.311, -140.938, 69.642, -195.767]
  Call Extruder(25649.571)
  MoveL 2732 to (-11.61, 24.12, 120) mm, rotated rx 180 ry 0 rz -180 deg; joints [36.473, 46.392, 18.84, -140.85, 70.312, -195.338]
  Call Extruder(25658.936)
  MoveL 2733 to (-16.69, 20.93, 120) mm, rotated rx 180 ry 0 rz -180 deg; joints [36.542, 45.616, 20.416, -140.957, 70.951, -194.826]
  Call Extruder(25668.302)
  MoveL 2734 to (-20.93, 16.69, 120) mm, rotated rx 180 ry 0 rz 180 deg; joints [36.407, 44.858, 21.959, -141.263, 71.529, -194.261]
  Call Extruder(25677.666)
  MoveL 2735 to (-24.12, 11.61, 120) mm, rotated rx -180 ry 0 rz -180 deg; joints [36.065, 44.155, 23.394, -141.761, 72.019, -193.672]
  Call Extruder(25687.031)
  MoveL 2736 to (-26.09, 5.96, 120) mm, rotated rx 180 ry 0 rz 180 deg; joints [35.528, 43.543, 24.647, -142.437, 72.401, -193.091]
  Call Extruder(25696.396)
  MoveL 2737 to (-26.77, 0, 120) mm, rotated rx -180 ry 0 rz 180 deg; joints [34.817, 43.053, 25.654, -143.262, 72.654, -192.546]
  Call Extruder(25701.185)
  MoveL 2738 to (-26.42, -3.05, 120) mm, rotated rx -180 ry 0 rz -180 deg; joints [34.385, 42.876, 26.018, -143.738, 72.712, -192.298]
  Set speed (130.0 mm/s)
  MoveL 2739 to (-41.86, -6.29, 120) mm, rotated rx 180 ry 0 rz 180 deg; joints [35.393, 41.129, 29.622, -143.036, 74.41, -191.434]
  Call Extruder(25706.183)
  Set speed (60.0 mm/s)
  MoveL 2740 to (-41.5, -9.47, 120) mm, rotated rx -180 ry 0 rz -180 deg; joints [34.924, 40.947, 29.999, -143.547, 74.474, -191.185]
  Call Extruder(25721.079)
  MoveL 2741 to (-38.36, -18.47, 120) mm, rotated rx 180 ry 0 rz -180 deg; joints [33.373, 40.66, 30.596, -145.177, 74.433, -190.574]
  Call Extruder(25735.974)
  MoveL 2742 to (-33.28, -26.54, 120) mm, rotated rx 180 ry 0 rz -180 deg; joints [31.763, 40.651, 30.613, -146.824, 74.151, -190.123]
  Call Extruder(25750.870)
  MoveL 2743 to (-26.54, -33.29, 120) mm, rotated rx -180 ry 0 rz 180 deg; joints [30.206, 40.923, 30.049, -148.375, 73.635, -189.843]
  Call Extruder(25765.766)
  MoveL 2744 to (-18.47, -38.36, 120) mm, rotated rx 180 ry 0 rz 180 deg; joints [28.808, 41.459, 28.939, -149.725, 72.904, -189.738]
  Call Extruder(25780.662)
  MoveL 2745 to (-9.47, -41.51, 120) mm, rotated rx 180 ry 0 rz 180 deg; joints [27.654, 42.231, 27.344, -150.789, 71.994, -189.806]
  Call Extruder(25795.558)
  MoveL 2746 to (0, -42.57, 120) mm, rotated rx 180 ry 0 rz 180 deg; joints [26.805, 43.198, 25.355, -151.506, 70.953, -190.046]
  Call Extruder(25807.926)
  MoveL 2747 to (7.87, -41.69, 120) mm, rotated rx 180 ry 0 rz -180 deg; joints [26.375, 44.12, 23.466, -151.791, 70.025, -190.383]
  Call Extruder(25810.454)
  MoveL 2748 to (9.47, -41.5, 120) mm, rotated rx 180 ry 0 rz 180 deg; joints [26.29, 44.311, 23.076, -151.846, 69.834, -190.453]
  Call Extruder(25825.349)
  MoveL 2749 to (18.47, -38.36, 120) mm, rotated rx 180 ry 0 rz 180 deg; joints [26.114, 45.514, 20.623, -151.808, 68.7, -191.018]
  Call Extruder(25840.245)
  MoveL 2750 to (26.54, -33.28, 120) mm, rotated rx 180 ry 0 rz 180 deg; joints [26.262, 46.748, 18.118, -151.41, 67.611, -191.727]
  Call Extruder(25855.141)
  MoveL 2751 to (33.28, -26.54, 120) mm, rotated rx 180 ry 0 rz -180 deg; joints [26.703, 47.952, 15.682, -150.689, 66.626, -192.557]
  Call Extruder(25870.037)
  MoveL 2752 to (38.36, -18.47, 120) mm, rotated rx 180 ry 0 rz 180 deg; joints [27.4, 49.069, 13.431, -149.699, 65.799, -193.472]
  Call Extruder(25884.932)
  MoveL 2753 to (41.5, -9.47, 120) mm, rotated rx 180 ry 0 rz -180 deg; joints [28.309, 50.043, 11.474, -148.499, 65.174, -194.429]
  Call Extruder(25899.828)
  MoveL 2754 to (42.57, 0, 120) mm, rotated rx 180 ry 0 rz 180 deg; joints [29.382, 50.824, 9.908, -147.159, 64.786, -195.375]
  Call Extruder(25914.724)
  MoveL 2755 to (41.5, 9.47, 120) mm, rotated rx 180 ry 0 rz 180 deg; joints [30.575, 51.373, 8.811, -145.747, 64.653, -196.252]
  Call Extruder(25929.620)
  MoveL 2756 to (38.36, 18.47, 120) mm, rotated rx 180 ry 0 rz 180 deg; joints [31.839, 51.659, 8.239, -144.33, 64.781, -197.005]
  Call Extruder(25944.516)
  MoveL 2757 to (33.29, 26.54, 120) mm, rotated rx 180 ry 0 rz -180 deg; joints [33.128, 51.667, 8.222, -142.97, 65.157, -197.585]
  Call Extruder(25959.411)
  MoveL 2758 to (26.54, 33.29, 120) mm, rotated rx 180 ry 0 rz -180 deg; joints [34.394, 51.397, 8.762, -141.719, 65.757, -197.955]
  Call Extruder(25974.307)
  MoveL 2759 to (18.47, 38.36, 120) mm, rotated rx -180 ry 0 rz -180 deg; joints [35.592, 50.864, 9.829, -140.621, 66.544, -198.093]
  Call Extruder(25989.203)
  MoveL 2760 to (9.47, 41.5, 120) mm, rotated rx -180 ry 0 rz 180 deg; joints [36.675, 50.095, 11.37, -139.714, 67.472, -197.992]
  Call Extruder(26004.099)
  MoveL 2761 to (0, 42.57, 120) mm, rotated rx 180 ry 0 rz -180 deg; joints [37.594, 49.131, 13.307, -139.026, 68.492, -197.663]
  Call Extruder(26018.995)
  MoveL 2762 to (-9.47, 41.5, 120) mm, rotated rx -180 ry 0 rz 180 deg; joints [38.304, 48.021, 15.543, -138.584, 69.552, -197.128]
  Call Extruder(26033.890)
  MoveL 2763 to (-18.47, 38.36, 120) mm, rotated rx 180 ry 0 rz -180 deg; joints [38.762, 46.82, 17.972, -138.412, 70.604, -196.422]
  Call Extruder(26048.786)
  MoveL 2764 to (-26.54, 33.29, 120) mm, rotated rx 180 ry 0 rz 180 deg; joints [38.928, 45.586, 20.476, -138.532, 71.6, -195.586]
  Call Extruder(26063.682)
  MoveL 2765 to (-33.29, 26.54, 120) mm, rotated rx 180 ry 0 rz -180 deg; joints [38.772, 44.38, 22.935, -138.958, 72.501, -194.669]
  Call Extruder(26078.578)
  MoveL 2766 to (-38.36, 18.47, 120) mm, rotated rx 180 ry 0 rz 180 deg; joints [38.277, 43.26, 25.228, -139.696, 73.27, -193.721]
  Call Extruder(26093.474)
  MoveL 2767 to (-41.5, 9.47, 120) mm, rotated rx 180 ry 0 rz 180 deg; joints [37.447, 42.283, 27.237, -140.733, 73.873, -192.794]
  Call Extruder(26108.369)
  MoveL 2768 to (-42.57, 0, 120) mm, rotated rx 180 ry 0 rz -180 deg; joints [36.31, 41.498, 28.857, -142.037, 74.282, -191.935]
  Call Extruder(26115.924)
  MoveL 2769 to (-42.03, -4.8, 120) mm, rotated rx 180 ry 0 rz 180 deg; joints [35.612, 41.215, 29.444, -142.798, 74.38, -191.551]
  Set speed (130.0 mm/s)
  MoveL 2770 to (-54.1, -7.67, 120) mm, rotated rx -180 ry 0 rz -180 deg; joints [36.421, 39.875, 32.229, -142.212, 75.684, -190.853]
  Call Extruder(26119.996)
  Set speed (30.0 mm/s)
  MoveL 2771 to (-53.59, -12.23, 120) mm, rotated rx -180 ry 0 rz -180 deg; joints [35.732, 39.614, 32.774, -142.955, 75.782, -190.503]
  Call Extruder(26130.926)
  MoveL 2772 to (-49.53, -23.85, 120) mm, rotated rx -180 ry 0 rz -180 deg; joints [33.663, 39.239, 33.558, -145.117, 75.749, -189.738]
  Call Extruder(26141.857)
  MoveL 2773 to (-42.98, -34.27, 120) mm, rotated rx 180 ry 0 rz 180 deg; joints [31.506, 39.228, 33.581, -147.316, 75.404, -189.184]
  Call Extruder(26152.787)
  MoveL 2774 to (-34.27, -42.98, 120) mm, rotated rx 180 ry 0 rz 180 deg; joints [29.427, 39.582, 32.841, -149.387, 74.75, -188.847]
  Call Extruder(26163.717)
  MoveL 2775 to (-23.85, -49.53, 120) mm, rotated rx -180 ry 0 rz 180 deg; joints [27.581, 40.28, 31.385, -151.176, 73.81, -188.723]
  Call Extruder(26174.647)
  MoveL 2776 to (-12.23, -53.59, 120) mm, rotated rx 180 ry 0 rz 180 deg; joints [26.087, 41.283, 29.304, -152.565, 72.631, -188.809]
  Call Extruder(26185.577)
  MoveL 2777 to (0, -54.97, 120) mm, rotated rx -180 ry 0 rz -180 deg; joints [25.019, 42.536, 26.716, -153.477, 71.275, -189.102]
  Call Extruder(26193.839)
  MoveL 2778 to (9.25, -53.93, 120) mm, rotated rx 180 ry 0 rz 180 deg; joints [24.552, 43.62, 24.49, -153.789, 70.177, -189.478]
  Call Extruder(26196.508)
  MoveL 2779 to (12.23, -53.59, 120) mm, rotated rx -180 ry 0 rz -180 deg; joints [24.406, 43.975, 23.762, -153.882, 69.818, -189.601]
  Call Extruder(26207.438)
  MoveL 2780 to (23.85, -49.52, 120) mm, rotated rx -180 ry 0 rz -180 deg; joints [24.239, 45.529, 20.593, -153.785, 68.339, -190.301]
  Call Extruder(26218.368)
  MoveL 2781 to (34.27, -42.98, 120) mm, rotated rx 180 ry 0 rz -180 deg; joints [24.487, 47.122, 17.361, -153.22, 66.919, -191.192]
  Call Extruder(26229.298)
  MoveL 2782 to (42.98, -34.27, 120) mm, rotated rx 180 ry 0 rz 180 deg; joints [25.101, 48.678, 14.218, -152.244, 65.633, -192.25]
  Call Extruder(26240.229)
  MoveL 2783 to (49.52, -23.85, 120) mm, rotated rx 180 ry 0 rz 180 deg; joints [26.025, 50.124, 11.313, -150.929, 64.554, -193.434]
  Call Extruder(26251.159)
  MoveL 2784 to (53.59, -12.23, 120) mm, rotated rx -180 ry 0 rz -180 deg; joints [27.2, 51.386, 8.783, -149.356, 63.741, -194.688]
  Call Extruder(26262.089)
  MoveL 2785 to (54.97, 0, 120) mm, rotated rx -180 ry 0 rz -180 deg; joints [28.57, 52.402, 6.753, -147.615, 63.239, -195.938]
  Call Extruder(26273.019)
  MoveL 2786 to (53.59, 12.23, 120) mm, rotated rx 180 ry 0 rz -180 deg; joints [30.077, 53.117, 5.329, -145.799, 63.074, -197.106]
  Call Extruder(26283.949)
  MoveL 2787 to (49.52, 23.85, 120) mm, rotated rx 180 ry 0 rz 180 deg; joints [31.665, 53.49, 4.585, -143.995, 63.251, -198.111]
  Call Extruder(26294.880)
  MoveL 2788 to (42.98, 34.27, 120) mm, rotated rx 180 ry 0 rz 180 deg; joints [33.282, 53.501, 4.564, -142.278, 63.756, -198.883]
  Call Extruder(26305.810)
  MoveL 2789 to (34.27, 42.98, 120) mm, rotated rx 180 ry 0 rz -180 deg; joints [34.874, 53.149, 5.266, -140.712, 64.551, -199.37]
  Call Extruder(26316.740)
  MoveL 2790 to (23.85, 49.53, 120) mm, rotated rx 180 ry 0 rz 180 deg; joints [36.387, 52.453, 6.652, -139.345, 65.584, -199.543]
  Call Extruder(26327.670)
  MoveL 2791 to (12.23, 53.59, 120) mm, rotated rx 180 ry 0 rz -180 deg; joints [37.766, 51.454, 8.648, -138.214, 66.794, -199.399]
  Call Extruder(26338.600)
  MoveL 2792 to (0, 54.97, 120) mm, rotated rx 180 ry 0 rz -180 deg; joints [38.954, 50.204, 11.152, -137.348, 68.113, -198.953]
  Call Extruder(26349.531)
  MoveL 2793 to (-12.23, 53.59, 120) mm, rotated rx 180 ry 0 rz 180 deg; joints [39.895, 48.767, 14.039, -136.776, 69.475, -198.239]
  Call Extruder(26360.461)
  MoveL 2794 to (-23.85, 49.52, 120) mm, rotated rx 180 ry 0 rz 180 deg; joints [40.528, 47.215, 17.172, -136.526, 70.818, -197.303]
  Call Extruder(26371.391)
  MoveL 2795 to (-34.27, 42.98, 120) mm, rotated rx 180 ry 0 rz 180 deg; joints [40.799, 45.622, 20.403, -136.63, 72.085, -196.203]
  Call Extruder(26382.321)
  MoveL 2796 to (-42.98, 34.27, 120) mm, rotated rx 180 ry 0 rz -180 deg; joints [40.659, 44.064, 23.58, -137.118, 73.23, -195]
  Call Extruder(26393.251)
  MoveL 2797 to (-49.53, 23.85, 120) mm, rotated rx 180 ry 0 rz 180 deg; joints [40.072, 42.616, 26.551, -138.01, 74.208, -193.764]
  Call Extruder(26404.181)
  MoveL 2798 to (-53.59, 12.23, 120) mm, rotated rx -180 ry 0 rz 180 deg; joints [39.031, 41.35, 29.164, -139.307, 74.982, -192.562]
  Call Extruder(26415.112)
  MoveL 2799 to (-54.97, 0, 120) mm, rotated rx -180 ry 0 rz 180 deg; joints [37.56, 40.331, 31.279, -140.979, 75.517, -191.457]
  Call Extruder(26420.637)
  MoveL 2800 to (-54.27, -6.18, 120) mm, rotated rx -180 ry 0 rz 180 deg; joints [36.644, 39.962, 32.047, -141.971, 75.652, -190.969]
  Set speed (130.0 mm/s)
  MoveL 2801 to (-49.9, -9.51, 120) mm, rotated rx 180 ry 0 rz 180 deg; joints [35.741, 40.143, 31.669, -142.856, 75.325, -190.864]
  MoveL 2802 to (2.97, -12.99, 120) mm, rotated rx -180 ry 0 rz 180 deg; joints [30.614, 45.309, 21.04, -147.138, 69.803, -192.573]
  Call Extruder(26425.301)
  Set speed (80.0 mm/s)
  MoveL 2803 to (5.78, -12.01, 120) mm, rotated rx -180 ry 0 rz 180 deg; joints [30.526, 45.685, 20.275, -147.151, 69.457, -192.766]
  Call Extruder(26429.965)
  MoveL 2804 to (8.31, -10.42, 120) mm, rotated rx 180 ry 0 rz 180 deg; joints [30.538, 46.072, 19.49, -147.056, 69.125, -193.002]
  Call Extruder(26434.629)
  MoveL 2805 to (10.42, -8.31, 120) mm, rotated rx 180 ry 0 rz 180 deg; joints [30.649, 46.449, 18.724, -146.86, 68.825, -193.27]
  Call Extruder(26439.292)
  MoveL 2806 to (12.01, -5.78, 120) mm, rotated rx 180 ry 0 rz -180 deg; joints [30.85, 46.798, 18.017, -146.573, 68.572, -193.558]
  Call Extruder(26443.956)
  MoveL 2807 to (12.99, -2.97, 120) mm, rotated rx 180 ry 0 rz 180 deg; joints [31.131, 47.101, 17.402, -146.212, 68.379, -193.85]
  Call Extruder(26448.620)
  MoveL 2808 to (13.33, 0, 120) mm, rotated rx -180 ry 0 rz -180 deg; joints [31.476, 47.344, 16.911, -145.797, 68.256, -194.133]
  Call Extruder(26453.284)
  MoveL 2809 to (12.99, 2.97, 120) mm, rotated rx 180 ry 0 rz 180 deg; joints [31.869, 47.514, 16.567, -145.347, 68.21, -194.391]
  Call Extruder(26457.947)
  MoveL 2810 to (12.01, 5.78, 120) mm, rotated rx 180 ry 0 rz 180 deg; joints [32.292, 47.602, 16.389, -144.886, 68.242, -194.61]
  Call Extruder(26462.611)
  MoveL 2811 to (10.42, 8.31, 120) mm, rotated rx 180 ry 0 rz 180 deg; joints [32.725, 47.605, 16.383, -144.434, 68.35, -194.778]
  Call Extruder(26467.275)
  MoveL 2812 to (8.31, 10.42, 120) mm, rotated rx -180 ry 0 rz -180 deg; joints [33.149, 47.522, 16.552, -144.013, 68.527, -194.887]
  Call Extruder(26471.939)
  MoveL 2813 to (5.78, 12.01, 120) mm, rotated rx -180 ry 0 rz -180 deg; joints [33.544, 47.356, 16.886, -143.642, 68.765, -194.929]
  Call Extruder(26476.602)
  MoveL 2814 to (2.97, 13, 120) mm, rotated rx 180 ry 0 rz -180 deg; joints [33.893, 47.117, 17.37, -143.337, 69.051, -194.903]
  Call Extruder(26481.266)
  MoveL 2815 to (0, 13.33, 120) mm, rotated rx 180 ry 0 rz 180 deg; joints [34.177, 46.817, 17.978, -143.113, 69.371, -194.81]
  Call Extruder(26485.930)
  MoveL 2816 to (-2.97, 13, 120) mm, rotated rx 180 ry 0 rz 180 deg; joints [34.384, 46.47, 18.681, -142.98, 69.708, -194.656]
  Call Extruder(26490.594)
  MoveL 2817 to (-5.78, 12.01, 120) mm, rotated rx 180 ry 0 rz -180 deg; joints [34.5, 46.094, 19.444, -142.945, 70.046, -194.449]
  Call Extruder(26495.257)
  MoveL 2818 to (-8.31, 10.42, 120) mm, rotated rx 180 ry 0 rz -180 deg; joints [34.518, 45.708, 20.229, -143.012, 70.369, -194.201]
  Call Extruder(26499.922)
  MoveL 2819 to (-10.42, 8.31, 120) mm, rotated rx -180 ry 0 rz 180 deg; joints [34.436, 45.331, 20.996, -143.18, 70.661, -193.924]
  Call Extruder(26504.585)
  MoveL 2820 to (-12.01, 5.78, 120) mm, rotated rx -180 ry 0 rz -180 deg; joints [34.254, 44.981, 21.708, -143.442, 70.908, -193.633]
  Call Extruder(26509.249)
  MoveL 2821 to (-13, 2.97, 120) mm, rotated rx 180 ry 0 rz 180 deg; joints [33.981, 44.677, 22.328, -143.788, 71.099, -193.343]
  Call Extruder(26513.913)
  MoveL 2822 to (-13.33, 0, 120) mm, rotated rx 180 ry 0 rz -180 deg; joints [33.63, 44.434, 22.825, -144.2, 71.224, -193.069]
  Call Extruder(26518.577)
  MoveL 2823 to (-13, -2.97, 120) mm, rotated rx -180 ry 0 rz -180 deg; joints [33.218, 44.263, 23.173, -144.66, 71.276, -192.823]
  Call Extruder(26523.240)
  MoveL 2824 to (-12.01, -5.78, 120) mm, rotated rx 180 ry 0 rz 180 deg; joints [32.767, 44.175, 23.355, -145.142, 71.253, -192.618]
  Call Extruder(26527.904)
  MoveL 2825 to (-10.42, -8.31, 120) mm, rotated rx 180 ry 0 rz 180 deg; joints [32.302, 44.172, 23.36, -145.621, 71.154, -192.462]
  Call Extruder(26532.568)
  MoveL 2826 to (-8.31, -10.42, 120) mm, rotated rx 180 ry 0 rz 180 deg; joints [31.85, 44.256, 23.189, -146.071, 70.985, -192.363]
  Call Extruder(26537.232)
  MoveL 2827 to (-5.78, -12.01, 120) mm, rotated rx 180 ry 0 rz 180 deg; joints [31.435, 44.422, 22.85, -146.467, 70.752, -192.324]
  Call Extruder(26541.895)
  MoveL 2828 to (-2.97, -12.99, 120) mm, rotated rx 180 ry 0 rz -180 deg; joints [31.079, 44.661, 22.361, -146.787, 70.468, -192.347]
  Call Extruder(26546.559)
  MoveL 2829 to (0, -13.33, 120) mm, rotated rx -180 ry 0 rz -180 deg; joints [30.801, 44.962, 21.748, -147.015, 70.146, -192.431]
  Call Extruder(26551.223)
  MoveL 2830 to (2.97, -12.99, 120) mm, rotated rx -180 ry 0 rz 180 deg; joints [30.614, 45.309, 21.04, -147.138, 69.803, -192.573]
  Set speed (130.0 mm/s)
  MoveL 2831 to (2.97, -13, 125) mm, rotated rx 180 ry 0 rz 180 deg; joints [30.614, 44.453, 21.234, -147.004, 69.248, -192.956]
  MoveL 2832 to (-26.25, -4.54, 125) mm, rotated rx 180 ry 0 rz 180 deg; joints [34.172, 41.891, 26.391, -143.842, 72.172, -192.611]
  Call Extruder(26553.456)
  Set speed (60.0 mm/s)
  MoveL 2833 to (-26.09, -5.96, 125) mm, rotated rx 180 ry 0 rz -180 deg; joints [33.969, 41.808, 26.557, -144.066, 72.196, -192.495]
  Call Extruder(26562.821)
  MoveL 2834 to (-24.12, -11.61, 125) mm, rotated rx 180 ry 0 rz 180 deg; joints [33.033, 41.626, 26.926, -145.061, 72.149, -192.088]
  Call Extruder(26572.186)
  MoveL 2835 to (-20.93, -16.69, 125) mm, rotated rx 180 ry 0 rz 180 deg; joints [32.066, 41.621, 26.937, -146.058, 71.953, -191.778]
  Call Extruder(26581.551)
  MoveL 2836 to (-16.69, -20.93, 125) mm, rotated rx -180 ry 0 rz 180 deg; joints [31.126, 41.793, 26.589, -146.994, 71.616, -191.577]
  Call Extruder(26590.916)
  MoveL 2837 to (-11.61, -24.11, 125) mm, rotated rx 180 ry 0 rz 180 deg; joints [30.272, 42.134, 25.901, -147.814, 71.153, -191.493]
  Call Extruder(26600.281)
  MoveL 2838 to (-5.96, -26.09, 125) mm, rotated rx 180 ry 0 rz -180 deg; joints [29.552, 42.625, 24.91, -148.47, 70.585, -191.527]
  Call Extruder(26609.646)
  MoveL 2839 to (0, -26.77, 125) mm, rotated rx -180 ry 0 rz -180 deg; joints [29.003, 43.241, 23.669, -148.924, 69.941, -191.679]
  Call Extruder(26619.011)
  MoveL 2840 to (5.96, -26.09, 125) mm, rotated rx -180 ry 0 rz -180 deg; joints [28.65, 43.951, 22.242, -149.156, 69.254, -191.944]
  Call Extruder(26628.376)
  MoveL 2841 to (11.61, -24.11, 125) mm, rotated rx 180 ry 0 rz 180 deg; joints [28.503, 44.719, 20.702, -149.158, 68.56, -192.313]
  Call Extruder(26637.740)
  MoveL 2842 to (16.69, -20.93, 125) mm, rotated rx 180 ry 0 rz -180 deg; joints [28.559, 45.507, 19.125, -148.936, 67.895, -192.772]
  Call Extruder(26647.106)
  MoveL 2843 to (20.93, -16.69, 125) mm, rotated rx 180 ry 0 rz 180 deg; joints [28.808, 46.275, 17.591, -148.51, 67.296, -193.302]
  Call Extruder(26656.471)
  MoveL 2844 to (24.11, -11.61, 125) mm, rotated rx 180 ry 0 rz -180 deg; joints [29.229, 46.986, 16.173, -147.908, 66.794, -193.88]
  Call Extruder(26665.835)
  MoveL 2845 to (26.09, -5.96, 125) mm, rotated rx 180 ry 0 rz 180 deg; joints [29.796, 47.604, 14.942, -147.166, 66.416, -194.476]
  Call Extruder(26675.200)
  MoveL 2846 to (26.77, 0, 125) mm, rotated rx -180 ry 0 rz 180 deg; joints [30.482, 48.099, 13.957, -146.325, 66.181, -195.06]
  Call Extruder(26684.566)
  MoveL 2847 to (26.09, 5.96, 125) mm, rotated rx 180 ry 0 rz 180 deg; joints [31.252, 48.445, 13.269, -145.427, 66.102, -195.599]
  Call Extruder(26693.930)
  MoveL 2848 to (24.11, 11.61, 125) mm, rotated rx 180 ry 0 rz 180 deg; joints [32.076, 48.625, 12.91, -144.516, 66.181, -196.061]
  Call Extruder(26703.295)
  MoveL 2849 to (20.93, 16.69, 125) mm, rotated rx 180 ry 0 rz 180 deg; joints [32.917, 48.631, 12.9, -143.632, 66.412, -196.419]
  Call Extruder(26712.661)
  MoveL 2850 to (16.69, 20.93, 125) mm, rotated rx 180 ry 0 rz 180 deg; joints [33.742, 48.46, 13.238, -142.813, 66.781, -196.652]
  Call Extruder(26722.025)
  MoveL 2851 to (11.61, 24.12, 125) mm, rotated rx 180 ry 0 rz -180 deg; joints [34.517, 48.123, 13.908, -142.093, 67.268, -196.746]
  Call Extruder(26731.390)
  MoveL 2852 to (5.96, 26.09, 125) mm, rotated rx 180 ry 0 rz -180 deg; joints [35.208, 47.637, 14.876, -141.5, 67.845, -196.698]
  Call Extruder(26740.755)
  MoveL 2853 to (0, 26.77, 125) mm, rotated rx 180 ry 0 rz -180 deg; joints [35.784, 47.025, 16.095, -141.058, 68.483, -196.51]
  Call Extruder(26750.120)
  MoveL 2854 to (-5.96, 26.09, 125) mm, rotated rx 180 ry 0 rz -180 deg; joints [36.214, 46.319, 17.503, -140.787, 69.149, -196.195]
  Call Extruder(26759.485)
  MoveL 2855 to (-11.61, 24.12, 125) mm, rotated rx 180 ry 0 rz -180 deg; joints [36.473, 45.553, 19.033, -140.702, 69.812, -195.772]
  Call Extruder(26768.850)
  MoveL 2856 to (-16.69, 20.93, 125) mm, rotated rx 180 ry 0 rz 180 deg; joints [36.542, 44.765, 20.609, -140.812, 70.441, -195.265]
  Call Extruder(26778.215)
  MoveL 2857 to (-20.93, 16.69, 125) mm, rotated rx 180 ry 0 rz -180 deg; joints [36.407, 43.995, 22.154, -141.121, 71.008, -194.703]
  Call Extruder(26787.580)
  MoveL 2858 to (-24.12, 11.61, 125) mm, rotated rx 180 ry 0 rz -180 deg; joints [36.065, 43.281, 23.59, -141.623, 71.486, -194.115]
  Call Extruder(26796.945)
  MoveL 2859 to (-26.09, 5.96, 125) mm, rotated rx 180 ry 0 rz -180 deg; joints [35.528, 42.658, 24.843, -142.301, 71.855, -193.533]
  Call Extruder(26806.310)
  MoveL 2860 to (-26.77, 0, 125) mm, rotated rx 180 ry 0 rz -180 deg; joints [34.817, 42.158, 25.851, -143.129, 72.096, -192.984]
  Call Extruder(26811.099)
  MoveL 2861 to (-26.42, -3.05, 125) mm, rotated rx 180 ry 0 rz -180 deg; joints [34.385, 41.978, 26.215, -143.607, 72.147, -192.733]
  Set speed (130.0 mm/s)
  MoveL 2862 to (-41.86, -6.29, 125) mm, rotated rx 180 ry 0 rz 180 deg; joints [35.393, 40.196, 29.823, -142.911, 73.826, -191.892]
  Call Extruder(26816.097)
  Set speed (60.0 mm/s)
  MoveL 2863 to (-41.5, -9.47, 125) mm, rotated rx 180 ry 0 rz -180 deg; joints [34.924, 40.011, 30.2, -143.423, 73.883, -191.639]
  Call Extruder(26830.992)
  MoveL 2864 to (-38.36, -18.47, 125) mm, rotated rx 180 ry 0 rz 180 deg; joints [33.373, 39.717, 30.797, -145.057, 73.825, -191.014]
  Call Extruder(26845.888)
  MoveL 2865 to (-33.29, -26.54, 125) mm, rotated rx 180 ry 0 rz 180 deg; joints [31.763, 39.709, 30.815, -146.707, 73.531, -190.546]
  Call Extruder(26860.784)
  MoveL 2866 to (-26.54, -33.28, 125) mm, rotated rx 180 ry 0 rz 180 deg; joints [30.206, 39.986, 30.251, -148.26, 73.009, -190.247]
  Call Extruder(26875.680)
  MoveL 2867 to (-18.47, -38.36, 125) mm, rotated rx 180 ry 0 rz 180 deg; joints [28.808, 40.533, 29.139, -149.611, 72.278, -190.122]
  Call Extruder(26890.576)
  MoveL 2868 to (-9.47, -41.51, 125) mm, rotated rx -180 ry 0 rz 180 deg; joints [27.654, 41.321, 27.543, -150.673, 71.374, -190.172]
  Call Extruder(26905.471)
  MoveL 2869 to (0, -42.57, 125) mm, rotated rx 180 ry 0 rz -180 deg; joints [26.805, 42.307, 25.552, -151.389, 70.342, -190.398]
  Call Extruder(26918.583)
  MoveL 2870 to (8.34, -41.63, 125) mm, rotated rx -180 ry 0 rz -180 deg; joints [26.35, 43.302, 23.546, -151.688, 69.371, -190.746]
  Call Extruder(26920.367)
  MoveL 2871 to (9.47, -41.5, 125) mm, rotated rx 180 ry 0 rz -180 deg; joints [26.29, 43.439, 23.271, -151.727, 69.238, -190.794]
  Call Extruder(26935.263)
  MoveL 2872 to (18.47, -38.36, 125) mm, rotated rx 180 ry 0 rz -180 deg; joints [26.114, 44.662, 20.817, -151.685, 68.12, -191.353]
  Call Extruder(26950.159)
  MoveL 2873 to (26.54, -33.28, 125) mm, rotated rx 180 ry 0 rz 180 deg; joints [26.262, 45.914, 18.311, -151.281, 67.048, -192.06]
  Call Extruder(26965.055)
  MoveL 2874 to (33.28, -26.54, 125) mm, rotated rx -180 ry 0 rz 180 deg; joints [26.703, 47.135, 15.874, -150.555, 66.082, -192.891]
  Call Extruder(26979.950)
  MoveL 2875 to (38.36, -18.47, 125) mm, rotated rx 180 ry 0 rz 180 deg; joints [27.4, 48.267, 13.623, -149.558, 65.272, -193.811]
  Call Extruder(26994.846)
  MoveL 2876 to (41.5, -9.47, 125) mm, rotated rx 180 ry 0 rz 180 deg; joints [28.309, 49.252, 11.666, -148.353, 64.664, -194.775]
  Call Extruder(27009.742)
  MoveL 2877 to (42.57, 0, 125) mm, rotated rx 180 ry 0 rz 180 deg; joints [29.382, 50.042, 10.1, -147.007, 64.291, -195.73]
  Call Extruder(27024.638)
  MoveL 2878 to (41.5, 9.47, 125) mm, rotated rx -180 ry 0 rz 180 deg; joints [30.575, 50.597, 9.003, -145.59, 64.171, -196.617]
  Call Extruder(27039.534)
  MoveL 2879 to (38.36, 18.47, 125) mm, rotated rx 180 ry 0 rz 180 deg; joints [31.839, 50.886, 8.431, -144.169, 64.31, -197.381]
  Call Extruder(27054.429)
  MoveL 2880 to (33.28, 26.54, 125) mm, rotated rx 180 ry 0 rz -180 deg; joints [33.128, 50.894, 8.415, -142.806, 64.695, -197.972]
  Call Extruder(27069.325)
  MoveL 2881 to (26.54, 33.29, 125) mm, rotated rx 180 ry 0 rz 180 deg; joints [34.394, 50.621, 8.954, -141.554, 65.3, -198.353]
  Call Extruder(27084.221)
  MoveL 2882 to (18.47, 38.36, 125) mm, rotated rx 180 ry 0 rz 180 deg; joints [35.592, 50.082, 10.022, -140.457, 66.089, -198.501]
  Call Extruder(27099.117)
  MoveL 2883 to (9.47, 41.51, 125) mm, rotated rx 180 ry 0 rz -180 deg; joints [36.675, 49.305, 11.563, -139.551, 67.017, -198.412]
  Call Extruder(27114.013)
  MoveL 2884 to (0, 42.57, 125) mm, rotated rx 180 ry 0 rz -180 deg; joints [37.594, 48.329, 13.499, -138.866, 68.032, -198.094]
  Call Extruder(27128.908)
  MoveL 2885 to (-9.47, 41.5, 125) mm, rotated rx -180 ry 0 rz 180 deg; joints [38.304, 47.205, 15.736, -138.428, 69.085, -197.569]
  Call Extruder(27143.804)
  MoveL 2886 to (-18.47, 38.36, 125) mm, rotated rx 180 ry 0 rz 180 deg; joints [38.762, 45.987, 18.165, -138.261, 70.126, -196.873]
  Call Extruder(27158.700)
  MoveL 2887 to (-26.54, 33.29, 125) mm, rotated rx 180 ry 0 rz -180 deg; joints [38.928, 44.735, 20.67, -138.385, 71.109, -196.046]
  Call Extruder(27173.596)
  MoveL 2888 to (-33.29, 26.54, 125) mm, rotated rx 180 ry 0 rz 180 deg; joints [38.772, 43.509, 23.13, -138.816, 71.992, -195.135]
  Call Extruder(27188.492)
  MoveL 2889 to (-38.36, 18.47, 125) mm, rotated rx -180 ry 0 rz 180 deg; joints [38.277, 42.37, 25.424, -139.558, 72.741, -194.191]
  Call Extruder(27203.387)
  MoveL 2890 to (-41.51, 9.47, 125) mm, rotated rx 180 ry 0 rz -180 deg; joints [37.447, 41.374, 27.436, -140.601, 73.323, -193.264]
  Call Extruder(27218.283)
  MoveL 2891 to (-42.57, 0, 125) mm, rotated rx 180 ry 0 rz 180 deg; joints [36.31, 40.573, 29.057, -141.909, 73.711, -192.4]
  Call Extruder(27225.837)
  MoveL 2892 to (-42.03, -4.8, 125) mm, rotated rx 180 ry 0 rz -180 deg; joints [35.612, 40.284, 29.644, -142.672, 73.799, -192.011]
  Set speed (130.0 mm/s)
  MoveL 2893 to (-54.1, -7.67, 125) mm, rotated rx 180 ry 0 rz 180 deg; joints [36.421, 38.915, 32.432, -142.091, 75.086, -191.333]
  Call Extruder(27229.910)
  Set speed (30.0 mm/s)
  MoveL 2894 to (-53.59, -12.23, 125) mm, rotated rx 180 ry 0 rz -180 deg; joints [35.732, 38.647, 32.979, -142.836, 75.174, -190.978]
  Call Extruder(27240.840)
  MoveL 2895 to (-49.53, -23.85, 125) mm, rotated rx 180 ry 0 rz 180 deg; joints [33.663, 38.263, 33.763, -145.002, 75.118, -190.194]
  Call Extruder(27251.771)
  MoveL 2896 to (-42.98, -34.27, 125) mm, rotated rx 180 ry 0 rz -180 deg; joints [31.506, 38.252, 33.786, -147.205, 74.757, -189.615]
  Call Extruder(27262.701)
  MoveL 2897 to (-34.27, -42.98, 125) mm, rotated rx 180 ry 0 rz 180 deg; joints [29.427, 38.615, 33.045, -149.278, 74.094, -189.25]
  Call Extruder(27273.631)
  MoveL 2898 to (-23.85, -49.52, 125) mm, rotated rx 180 ry 0 rz 180 deg; joints [27.581, 39.329, 31.588, -151.069, 73.155, -189.1]
  Call Extruder(27284.561)
  MoveL 2899 to (-12.23, -53.59, 125) mm, rotated rx 180 ry 0 rz 180 deg; joints [26.087, 40.353, 29.504, -152.458, 71.984, -189.162]
  Call Extruder(27295.491)
  MoveL 2900 to (0, -54.97, 125) mm, rotated rx 180 ry 0 rz -180 deg; joints [25.019, 41.632, 26.914, -153.368, 70.644, -189.436]
  Call Extruder(27304.175)
  MoveL 2901 to (9.72, -53.87, 125) mm, rotated rx 180 ry 0 rz 180 deg; joints [24.528, 42.793, 24.571, -153.692, 69.504, -189.821]
  Call Extruder(27306.421)
  MoveL 2902 to (12.23, -53.59, 125) mm, rotated rx 180 ry 0 rz 180 deg; joints [24.406, 43.098, 23.958, -153.77, 69.206, -189.922]
  Call Extruder(27317.352)
  MoveL 2903 to (23.85, -49.52, 125) mm, rotated rx 180 ry 0 rz 180 deg; joints [24.239, 44.677, 20.787, -153.667, 67.749, -190.615]
  Call Extruder(27328.282)
  MoveL 2904 to (34.27, -42.98, 125) mm, rotated rx 180 ry 0 rz 180 deg; joints [24.487, 46.293, 17.554, -153.096, 66.352, -191.505]
  Call Extruder(27339.212)
  MoveL 2905 to (42.98, -34.27, 125) mm, rotated rx -180 ry 0 rz 180 deg; joints [25.101, 47.871, 14.411, -152.113, 65.089, -192.566]
  Call Extruder(27350.142)
  MoveL 2906 to (49.52, -23.85, 125) mm, rotated rx 180 ry 0 rz -180 deg; joints [26.025, 49.334, 11.505, -150.789, 64.032, -193.757]
  Call Extruder(27361.072)
  MoveL 2907 to (53.59, -12.23, 125) mm, rotated rx 180 ry 0 rz -180 deg; joints [27.2, 50.611, 8.976, -149.207, 63.24, -195.02]
  Call Extruder(27372.003)
  MoveL 2908 to (54.97, 0, 125) mm, rotated rx 180 ry 0 rz -180 deg; joints [28.57, 51.637, 6.947, -147.459, 62.756, -196.283]
  Call Extruder(27382.933)
  MoveL 2909 to (53.59, 12.23, 125) mm, rotated rx 180 ry 0 rz -180 deg; joints [30.077, 52.358, 5.523, -145.636, 62.607, -197.464]
  Call Extruder(27393.863)
  MoveL 2910 to (49.52, 23.85, 125) mm, rotated rx 180 ry 0 rz 180 deg; joints [31.665, 52.735, 4.78, -143.827, 62.798, -198.482]
  Call Extruder(27404.793)
  MoveL 2911 to (42.98, 34.27, 125) mm, rotated rx -180 ry 0 rz -180 deg; joints [33.282, 52.746, 4.758, -142.107, 63.313, -199.267]
  Call Extruder(27415.723)
  MoveL 2912 to (34.27, 42.98, 125) mm, rotated rx 180 ry 0 rz 180 deg; joints [34.874, 52.39, 5.46, -140.54, 64.115, -199.767]
  Call Extruder(27426.654)
  MoveL 2913 to (23.85, 49.53, 125) mm, rotated rx 180 ry 0 rz 180 deg; joints [36.387, 51.688, 6.845, -139.174, 65.151, -199.954]
  Call Extruder(27437.584)
  MoveL 2914 to (12.23, 53.59, 125) mm, rotated rx 180 ry 0 rz 180 deg; joints [37.766, 50.679, 8.841, -138.046, 66.36, -199.823]
  Call Extruder(27448.514)
  MoveL 2915 to (0, 54.97, 125) mm, rotated rx -180 ry 0 rz 180 deg; joints [38.954, 49.415, 11.345, -137.184, 67.675, -199.39]
  Call Extruder(27459.444)
  MoveL 2916 to (-12.23, 53.59, 125) mm, rotated rx 180 ry 0 rz 180 deg; joints [39.895, 47.961, 14.232, -136.616, 69.028, -198.689]
  Call Extruder(27470.374)
  MoveL 2917 to (-23.85, 49.52, 125) mm, rotated rx 180 ry 0 rz 180 deg; joints [40.528, 46.388, 17.365, -136.372, 70.358, -197.767]
  Call Extruder(27481.305)
  MoveL 2918 to (-34.27, 42.98, 125) mm, rotated rx -180 ry 0 rz -180 deg; joints [40.799, 44.772, 20.597, -136.482, 71.609, -196.678]
  Call Extruder(27492.235)
  MoveL 2919 to (-42.98, 34.27, 125) mm, rotated rx 180 ry 0 rz 180 deg; joints [40.659, 43.188, 23.776, -136.976, 72.731, -195.485]
  Call Extruder(27503.165)
  MoveL 2920 to (-49.53, 23.85, 125) mm, rotated rx 180 ry 0 rz -180 deg; joints [40.072, 41.714, 26.749, -137.874, 73.685, -194.255]
  Call Extruder(27514.095)
  MoveL 2921 to (-53.59, 12.23, 125) mm, rotated rx 180 ry 0 rz 180 deg; joints [39.031, 40.422, 29.364, -139.177, 74.431, -193.054]
  Call Extruder(27525.025)
  MoveL 2922 to (-54.97, 0, 125) mm, rotated rx 180 ry 0 rz -180 deg; joints [37.56, 39.381, 31.482, -140.855, 74.937, -191.944]
  Call Extruder(27530.551)
  MoveL 2923 to (-54.27, -6.18, 125) mm, rotated rx -180 ry 0 rz -180 deg; joints [36.644, 39.004, 32.251, -141.849, 75.057, -191.45]
  Set speed (130.0 mm/s)
  MoveL 2924 to (-49.9, -9.51, 125) mm, rotated rx 180 ry 0 rz 180 deg; joints [35.741, 39.189, 31.872, -142.734, 74.726, -191.334]
  MoveL 2925 to (2.97, -13, 125) mm, rotated rx 180 ry 0 rz 180 deg; joints [30.614, 44.453, 21.234, -147.004, 69.248, -192.956]
  Call Extruder(27535.215)
  Set speed (80.0 mm/s)
  MoveL 2926 to (5.78, -12.01, 125) mm, rotated rx -180 ry 0 rz 180 deg; joints [30.526, 44.836, 20.469, -147.016, 68.906, -193.147]
  Call Extruder(27539.878)
  MoveL 2927 to (8.31, -10.42, 125) mm, rotated rx 180 ry 0 rz -180 deg; joints [30.538, 45.228, 19.683, -146.919, 68.58, -193.382]
  Call Extruder(27544.542)
  MoveL 2928 to (10.42, -8.31, 125) mm, rotated rx 180 ry 0 rz 180 deg; joints [30.649, 45.611, 18.918, -146.721, 68.285, -193.65]
  Call Extruder(27549.206)
  MoveL 2929 to (12.01, -5.78, 125) mm, rotated rx 180 ry 0 rz 180 deg; joints [30.85, 45.965, 18.21, -146.432, 68.038, -193.938]
  Call Extruder(27553.870)
  MoveL 2930 to (12.99, -2.97, 125) mm, rotated rx -180 ry 0 rz -180 deg; joints [31.131, 46.273, 17.595, -146.07, 67.851, -194.232]
  Call Extruder(27558.534)
  MoveL 2931 to (13.33, 0, 125) mm, rotated rx -180 ry 0 rz -180 deg; joints [31.476, 46.519, 17.104, -145.653, 67.734, -194.517]
  Call Extruder(27563.198)
  MoveL 2932 to (12.99, 2.97, 125) mm, rotated rx -180 ry 0 rz 180 deg; joints [31.869, 46.691, 16.76, -145.202, 67.692, -194.778]
  Call Extruder(27567.861)
  MoveL 2933 to (12.01, 5.78, 125) mm, rotated rx 180 ry 0 rz -180 deg; joints [32.292, 46.781, 16.581, -144.739, 67.728, -195.001]
  Call Extruder(27572.525)
  MoveL 2934 to (10.42, 8.31, 125) mm, rotated rx 180 ry 0 rz 180 deg; joints [32.725, 46.783, 16.576, -144.286, 67.838, -195.173]
  Call Extruder(27577.189)
  MoveL 2935 to (8.31, 10.42, 125) mm, rotated rx 180 ry 0 rz -180 deg; joints [33.149, 46.699, 16.745, -143.865, 68.018, -195.286]
  Call Extruder(27581.853)
  MoveL 2936 to (5.78, 12.01, 125) mm, rotated rx 180 ry 0 rz -180 deg; joints [33.544, 46.531, 17.079, -143.494, 68.257, -195.333]
  Call Extruder(27586.516)
  MoveL 2937 to (2.97, 12.99, 125) mm, rotated rx -180 ry 0 rz 180 deg; joints [33.893, 46.289, 17.562, -143.189, 68.542, -195.311]
  Call Extruder(27591.180)
  MoveL 2938 to (0, 13.33, 125) mm, rotated rx -180 ry 0 rz -180 deg; joints [34.177, 45.984, 18.171, -142.966, 68.86, -195.222]
  Call Extruder(27595.844)
  MoveL 2939 to (-2.97, 12.99, 125) mm, rotated rx 180 ry 0 rz 180 deg; joints [34.384, 45.632, 18.874, -142.834, 69.194, -195.071]
  Call Extruder(27600.508)
  MoveL 2940 to (-5.78, 12.01, 125) mm, rotated rx -180 ry 0 rz -180 deg; joints [34.5, 45.251, 19.637, -142.801, 69.528, -194.867]
  Call Extruder(27605.171)
  MoveL 2941 to (-8.31, 10.42, 125) mm, rotated rx 180 ry 0 rz 180 deg; joints [34.518, 44.859, 20.423, -142.87, 69.846, -194.621]
  Call Extruder(27609.835)
  MoveL 2942 to (-10.42, 8.31, 125) mm, rotated rx 180 ry 0 rz -180 deg; joints [34.436, 44.475, 21.19, -143.039, 70.132, -194.345]
  Call Extruder(27614.499)
  MoveL 2943 to (-12.01, 5.78, 125) mm, rotated rx 180 ry 0 rz 180 deg; joints [34.254, 44.12, 21.903, -143.303, 70.374, -194.054]
  Call Extruder(27619.163)
  MoveL 2944 to (-13, 2.97, 125) mm, rotated rx -180 ry 0 rz -180 deg; joints [33.981, 43.811, 22.523, -143.65, 70.558, -193.764]
  Call Extruder(27623.827)
  MoveL 2945 to (-13.33, 0, 125) mm, rotated rx 180 ry 0 rz 180 deg; joints [33.63, 43.564, 23.02, -144.064, 70.677, -193.487]
  Call Extruder(27628.491)
  MoveL 2946 to (-13, -2.97, 125) mm, rotated rx 180 ry 0 rz -180 deg; joints [33.218, 43.391, 23.369, -144.524, 70.724, -193.239]
  Call Extruder(27633.154)
  MoveL 2947 to (-12.01, -5.78, 125) mm, rotated rx 180 ry 0 rz -180 deg; joints [32.767, 43.3, 23.55, -145.008, 70.696, -193.029]
  Call Extruder(27637.818)
  MoveL 2948 to (-10.42, -8.31, 125) mm, rotated rx 180 ry 0 rz -180 deg; joints [32.302, 43.298, 23.555, -145.488, 70.594, -192.869]
  Call Extruder(27642.482)
  MoveL 2949 to (-8.31, -10.42, 125) mm, rotated rx -180 ry 0 rz -180 deg; joints [31.85, 43.383, 23.384, -145.939, 70.423, -192.764]
  Call Extruder(27647.146)
  MoveL 2950 to (-5.78, -12.01, 125) mm, rotated rx -180 ry 0 rz -180 deg; joints [31.435, 43.551, 23.045, -146.335, 70.19, -192.72]
  Call Extruder(27651.809)
  MoveL 2951 to (-2.97, -12.99, 125) mm, rotated rx 180 ry 0 rz 180 deg; joints [31.079, 43.795, 22.556, -146.655, 69.907, -192.738]
  Call Extruder(27656.473)
  MoveL 2952 to (0, -13.33, 125) mm, rotated rx -180 ry 0 rz -180 deg; joints [30.801, 44.101, 21.942, -146.881, 69.587, -192.818]
  Call Extruder(27661.137)
  MoveL 2953 to (2.97, -13, 125) mm, rotated rx 180 ry 0 rz 180 deg; joints [30.614, 44.453, 21.234, -147.004, 69.248, -192.956]
  Set speed (130.0 mm/s)
  MoveL 2954 to (2.97, -12.99, 130) mm, rotated rx 180 ry 0 rz 180 deg; joints [30.614, 43.605, 21.411, -146.863, 68.685, -193.349]
  MoveL 2955 to (-26.25, -4.54, 130) mm, rotated rx 180 ry 0 rz 180 deg; joints [34.172, 40.999, 26.571, -143.704, 71.598, -193.054]
  Call Extruder(27663.370)
  Set speed (60.0 mm/s)
  MoveL 2956 to (-26.09, -5.96, 130) mm, rotated rx 180 ry 0 rz 180 deg; joints [33.969, 40.915, 26.738, -143.929, 71.619, -192.937]
  Call Extruder(27672.734)
  MoveL 2957 to (-24.12, -11.61, 130) mm, rotated rx -180 ry 0 rz 180 deg; joints [33.033, 40.729, 27.107, -144.927, 71.562, -192.52]
  Call Extruder(27682.099)
  MoveL 2958 to (-20.93, -16.69, 130) mm, rotated rx 180 ry 0 rz 180 deg; joints [32.066, 40.723, 27.117, -145.925, 71.359, -192.2]
  Call Extruder(27691.465)
  MoveL 2959 to (-16.69, -20.93, 130) mm, rotated rx 180 ry 0 rz -180 deg; joints [31.126, 40.899, 26.769, -146.862, 71.018, -191.988]
  Call Extruder(27700.830)
  MoveL 2960 to (-11.61, -24.11, 130) mm, rotated rx -180 ry 0 rz -180 deg; joints [30.272, 41.246, 26.081, -147.683, 70.554, -191.893]
  Call Extruder(27710.194)
  MoveL 2961 to (-5.96, -26.09, 130) mm, rotated rx 180 ry 0 rz -180 deg; joints [29.552, 41.746, 25.089, -148.338, 69.989, -191.916]
  Call Extruder(27719.559)
  MoveL 2962 to (0, -26.77, 130) mm, rotated rx 180 ry 0 rz -180 deg; joints [29.003, 42.373, 23.847, -148.792, 69.35, -192.059]
  Call Extruder(27728.925)
  MoveL 2963 to (5.96, -26.09, 130) mm, rotated rx 180 ry 0 rz -180 deg; joints [28.65, 43.095, 22.42, -149.022, 68.671, -192.318]
  Call Extruder(27738.289)
  MoveL 2964 to (11.61, -24.11, 130) mm, rotated rx 180 ry 0 rz -180 deg; joints [28.503, 43.875, 20.879, -149.021, 67.987, -192.682]
  Call Extruder(27747.654)
  MoveL 2965 to (16.69, -20.93, 130) mm, rotated rx 180 ry 0 rz -180 deg; joints [28.559, 44.674, 19.302, -148.796, 67.334, -193.139]
  Call Extruder(27757.019)
  MoveL 2966 to (20.93, -16.69, 130) mm, rotated rx 180 ry 0 rz 180 deg; joints [28.808, 45.453, 17.766, -148.367, 66.746, -193.669]
  Call Extruder(27766.384)
  MoveL 2967 to (24.12, -11.61, 130) mm, rotated rx -180 ry 0 rz -180 deg; joints [29.229, 46.174, 16.348, -147.761, 66.256, -194.249]
  Call Extruder(27775.749)
  MoveL 2968 to (26.09, -5.96, 130) mm, rotated rx 180 ry 0 rz 180 deg; joints [29.796, 46.8, 15.117, -147.015, 65.889, -194.85]
  Call Extruder(27785.114)
  MoveL 2969 to (26.77, 0, 130) mm, rotated rx 180 ry 0 rz -180 deg; joints [30.482, 47.302, 14.132, -146.17, 65.664, -195.439]
  Call Extruder(27794.479)
  MoveL 2970 to (26.09, 5.96, 130) mm, rotated rx 180 ry 0 rz -180 deg; joints [31.252, 47.652, 13.444, -145.269, 65.594, -195.984]
  Call Extruder(27803.844)
  MoveL 2971 to (24.11, 11.61, 130) mm, rotated rx -180 ry 0 rz -180 deg; joints [32.076, 47.835, 13.086, -144.356, 65.68, -196.453]
  Call Extruder(27813.209)
  MoveL 2972 to (20.93, 16.69, 130) mm, rotated rx 180 ry 0 rz 180 deg; joints [32.917, 47.84, 13.075, -143.47, 65.917, -196.819]
  Call Extruder(27822.574)
  MoveL 2973 to (16.69, 20.93, 130) mm, rotated rx 180 ry 0 rz 180 deg; joints [33.742, 47.668, 13.414, -142.651, 66.29, -197.06]
  Call Extruder(27831.939)
  MoveL 2974 to (11.61, 24.11, 130) mm, rotated rx -180 ry 0 rz 180 deg; joints [34.517, 47.326, 14.083, -141.931, 66.778, -197.162]
  Call Extruder(27841.304)
  MoveL 2975 to (5.96, 26.09, 130) mm, rotated rx 180 ry 0 rz -180 deg; joints [35.208, 46.834, 15.051, -141.339, 67.354, -197.121]
  Call Extruder(27850.669)
  MoveL 2976 to (0, 26.77, 130) mm, rotated rx -180 ry 0 rz -180 deg; joints [35.784, 46.214, 16.27, -140.898, 67.989, -196.941]
  Call Extruder(27860.034)
  MoveL 2977 to (-5.96, 26.09, 130) mm, rotated rx 180 ry 0 rz -180 deg; joints [36.214, 45.498, 17.679, -140.629, 68.65, -196.633]
  Call Extruder(27869.399)
  MoveL 2978 to (-11.61, 24.12, 130) mm, rotated rx 180 ry 0 rz -180 deg; joints [36.473, 44.721, 19.209, -140.547, 69.305, -196.216]
  Call Extruder(27878.764)
  MoveL 2979 to (-16.69, 20.93, 130) mm, rotated rx 180 ry 0 rz 180 deg; joints [36.542, 43.922, 20.786, -140.66, 69.925, -195.714]
  Call Extruder(27888.129)
  MoveL 2980 to (-20.93, 16.69, 130) mm, rotated rx 180 ry 0 rz 180 deg; joints [36.407, 43.139, 22.331, -140.972, 70.48, -195.155]
  Call Extruder(27897.494)
  MoveL 2981 to (-24.11, 11.61, 130) mm, rotated rx 180 ry 0 rz -180 deg; joints [36.065, 42.413, 23.768, -141.477, 70.947, -194.568]
  Call Extruder(27906.859)
  MoveL 2982 to (-26.09, 5.96, 130) mm, rotated rx 180 ry 0 rz -180 deg; joints [35.528, 41.78, 25.022, -142.159, 71.302, -193.984]
  Call Extruder(27916.224)
  MoveL 2983 to (-26.77, 0, 130) mm, rotated rx 180 ry 0 rz -180 deg; joints [34.817, 41.271, 26.03, -142.989, 71.53, -193.432]
  Call Extruder(27921.013)
  MoveL 2984 to (-26.42, -3.05, 130) mm, rotated rx -180 ry 0 rz -180 deg; joints [34.385, 41.087, 26.395, -143.469, 71.576, -193.177]
  Set speed (130.0 mm/s)
  MoveL 2985 to (-41.86, -6.29, 130) mm, rotated rx 180 ry 0 rz 180 deg; joints [35.393, 39.271, 30.006, -142.779, 73.234, -192.36]
  Call Extruder(27926.011)
  Set speed (60.0 mm/s)
  MoveL 2986 to (-41.5, -9.47, 130) mm, rotated rx 180 ry 0 rz -180 deg; joints [34.924, 39.081, 30.383, -143.291, 73.285, -192.104]
  Call Extruder(27940.906)
  MoveL 2987 to (-38.36, -18.47, 130) mm, rotated rx 180 ry 0 rz 180 deg; joints [33.373, 38.781, 30.981, -144.929, 73.21, -191.464]
  Call Extruder(27955.802)
  MoveL 2988 to (-33.28, -26.54, 130) mm, rotated rx 180 ry 0 rz 180 deg; joints [31.763, 38.773, 30.999, -146.582, 72.903, -190.978]
  Call Extruder(27970.698)
  MoveL 2989 to (-26.54, -33.28, 130) mm, rotated rx 180 ry 0 rz 180 deg; joints [30.206, 39.056, 30.434, -148.137, 72.374, -190.659]
  Call Extruder(27985.594)
  MoveL 2990 to (-18.47, -38.36, 130) mm, rotated rx 180 ry 0 rz -180 deg; joints [28.808, 39.615, 29.321, -149.489, 71.643, -190.514]
  Call Extruder(28000.489)
  MoveL 2991 to (-9.47, -41.5, 130) mm, rotated rx 180 ry 0 rz 180 deg; joints [27.654, 40.418, 27.724, -150.552, 70.744, -190.547]
  Call Extruder(28015.385)
  MoveL 2992 to (0, -42.57, 130) mm, rotated rx 180 ry 0 rz -180 deg; joints [26.805, 41.422, 25.731, -151.266, 69.724, -190.758]
  Call Extruder(28029.065)
  MoveL 2993 to (8.7, -41.59, 130) mm, rotated rx -180 ry 0 rz 180 deg; joints [26.331, 42.479, 23.637, -151.576, 68.723, -191.112]
  Call Extruder(28030.281)
  MoveL 2994 to (9.47, -41.5, 130) mm, rotated rx 180 ry 0 rz 180 deg; joints [26.29, 42.574, 23.449, -151.601, 68.633, -191.144]
  Call Extruder(28045.177)
  MoveL 2995 to (18.47, -38.36, 130) mm, rotated rx 180 ry 0 rz 180 deg; joints [26.114, 43.817, 20.994, -151.555, 67.532, -191.696]
  Call Extruder(28060.073)
  MoveL 2996 to (26.54, -33.28, 130) mm, rotated rx 180 ry 0 rz -180 deg; joints [26.262, 45.088, 18.487, -151.147, 66.478, -192.401]
  Call Extruder(28074.968)
  MoveL 2997 to (33.28, -26.54, 130) mm, rotated rx 180 ry 0 rz 180 deg; joints [26.703, 46.326, 16.05, -150.415, 65.53, -193.234]
  Call Extruder(28089.864)
  MoveL 2998 to (38.36, -18.47, 130) mm, rotated rx 180 ry 0 rz -180 deg; joints [27.4, 47.472, 13.798, -149.412, 64.738, -194.158]
  Call Extruder(28104.760)
  MoveL 2999 to (41.5, -9.47, 130) mm, rotated rx -180 ry 0 rz 180 deg; joints [28.309, 48.469, 11.842, -148.2, 64.147, -195.13]
  Call Extruder(28119.656)
  MoveL 3000 to (42.57, 0, 130) mm, rotated rx 180 ry 0 rz 180 deg; joints [29.382, 49.268, 10.275, -146.847, 63.789, -196.093]
  Call Extruder(28134.552)
  MoveL 3001 to (41.5, 9.47, 130) mm, rotated rx 180 ry 0 rz -180 deg; joints [30.575, 49.828, 9.179, -145.425, 63.683, -196.991]
  Call Extruder(28149.447)
  MoveL 3002 to (38.36, 18.47, 130) mm, rotated rx -180 ry 0 rz -180 deg; joints [31.839, 50.12, 8.607, -144.001, 63.832, -197.765]
  Call Extruder(28164.343)
  MoveL 3003 to (33.29, 26.54, 130) mm, rotated rx 180 ry 0 rz 180 deg; joints [33.128, 50.129, 8.591, -142.635, 64.225, -198.368]
  Call Extruder(28179.239)
  MoveL 3004 to (26.54, 33.29, 130) mm, rotated rx 180 ry 0 rz 180 deg; joints [34.394, 49.853, 9.13, -141.383, 64.837, -198.76]
  Call Extruder(28194.135)
  MoveL 3005 to (18.47, 38.36, 130) mm, rotated rx 180 ry 0 rz 180 deg; joints [35.592, 49.308, 10.197, -140.286, 65.628, -198.92]
  Call Extruder(28209.031)
  MoveL 3006 to (9.47, 41.51, 130) mm, rotated rx 180 ry 0 rz 180 deg; joints [36.675, 48.522, 11.738, -139.382, 66.555, -198.841]
  Call Extruder(28223.926)
  MoveL 3007 to (0, 42.57, 130) mm, rotated rx 180 ry 0 rz -180 deg; joints [37.594, 47.535, 13.674, -138.699, 67.566, -198.534]
  Call Extruder(28238.822)
  MoveL 3008 to (-9.47, 41.51, 130) mm, rotated rx 180 ry 0 rz -180 deg; joints [38.304, 46.396, 15.911, -138.265, 68.612, -198.021]
  Call Extruder(28253.718)
  MoveL 3009 to (-18.47, 38.36, 130) mm, rotated rx 180 ry 0 rz -180 deg; joints [38.762, 45.162, 18.341, -138.102, 69.642, -197.334]
  Call Extruder(28268.614)
  MoveL 3010 to (-26.54, 33.28, 130) mm, rotated rx -180 ry 0 rz -180 deg; joints [38.928, 43.891, 20.847, -138.231, 70.61, -196.516]
  Call Extruder(28283.510)
  MoveL 3011 to (-33.29, 26.54, 130) mm, rotated rx -180 ry 0 rz -180 deg; joints [38.772, 42.645, 23.308, -138.667, 71.477, -195.612]
  Call Extruder(28298.405)
  MoveL 3012 to (-38.36, 18.47, 130) mm, rotated rx 180 ry 0 rz -180 deg; joints [38.277, 41.486, 25.604, -139.414, 72.206, -194.671]
  Call Extruder(28313.301)
  MoveL 3013 to (-41.5, 9.47, 130) mm, rotated rx 180 ry 0 rz -180 deg; joints [37.447, 40.472, 27.616, -140.461, 72.766, -193.743]
  Call Extruder(28328.197)
  MoveL 3014 to (-42.57, 0, 130) mm, rotated rx 180 ry 0 rz 180 deg; joints [36.31, 39.656, 29.24, -141.773, 73.133, -192.874]
  Call Extruder(28335.751)
  MoveL 3015 to (-42.03, -4.8, 130) mm, rotated rx -180 ry 0 rz -180 deg; joints [35.612, 39.361, 29.827, -142.539, 73.21, -192.48]
  Set speed (130.0 mm/s)
  MoveL 3016 to (-54.1, -7.67, 130) mm, rotated rx 180 ry 0 rz -180 deg; joints [36.421, 37.961, 32.618, -141.962, 74.481, -191.823]
  Call Extruder(28339.824)
  Set speed (30.0 mm/s)
  MoveL 3017 to (-53.59, -12.23, 130) mm, rotated rx 180 ry 0 rz 180 deg; joints [35.732, 37.688, 33.165, -142.709, 74.558, -191.462]
  Call Extruder(28350.754)
  MoveL 3018 to (-49.52, -23.85, 130) mm, rotated rx 180 ry 0 rz -180 deg; joints [33.663, 37.295, 33.951, -144.88, 74.479, -190.659]
  Call Extruder(28361.684)
  MoveL 3019 to (-42.98, -34.27, 130) mm, rotated rx 180 ry 0 rz -180 deg; joints [31.506, 37.283, 33.973, -147.087, 74.1, -190.055]
  Call Extruder(28372.614)
  MoveL 3020 to (-34.27, -42.98, 130) mm, rotated rx 180 ry 0 rz 180 deg; joints [29.427, 37.654, 33.232, -149.163, 73.429, -189.663]
  Call Extruder(28383.545)
  MoveL 3021 to (-23.85, -49.53, 130) mm, rotated rx 180 ry 0 rz 180 deg; joints [27.581, 38.384, 31.773, -150.955, 72.491, -189.485]
  Call Extruder(28394.475)
  MoveL 3022 to (-12.23, -53.59, 130) mm, rotated rx 180 ry 0 rz 180 deg; joints [26.087, 39.431, 29.687, -152.344, 71.329, -189.523]
  Call Extruder(28405.405)
  MoveL 3023 to (0, -54.97, 130) mm, rotated rx 180 ry 0 rz 180 deg; joints [25.019, 40.735, 27.094, -153.253, 70.004, -189.778]
  Call Extruder(28414.412)
  MoveL 3024 to (10.08, -53.83, 130) mm, rotated rx -180 ry 0 rz -180 deg; joints [24.511, 41.961, 24.662, -153.585, 68.837, -190.166]
  Call Extruder(28416.335)
  MoveL 3025 to (12.23, -53.59, 130) mm, rotated rx 180 ry 0 rz -180 deg; joints [24.406, 42.227, 24.136, -153.651, 68.586, -190.25]
  Call Extruder(28427.265)
  MoveL 3026 to (23.85, -49.52, 130) mm, rotated rx -180 ry 0 rz -180 deg; joints [24.239, 43.832, 20.963, -153.544, 67.151, -190.937]
  Call Extruder(28438.196)
  MoveL 3027 to (34.27, -42.98, 130) mm, rotated rx -180 ry 0 rz 180 deg; joints [24.487, 45.472, 17.729, -152.966, 65.776, -191.825]
  Call Extruder(28449.126)
  MoveL 3028 to (42.98, -34.27, 130) mm, rotated rx 180 ry 0 rz 180 deg; joints [25.101, 47.071, 14.586, -151.975, 64.537, -192.889]
  Call Extruder(28460.056)
  MoveL 3029 to (49.52, -23.85, 130) mm, rotated rx 180 ry 0 rz -180 deg; joints [26.025, 48.551, 11.68, -150.642, 63.503, -194.088]
  Call Extruder(28470.986)
  MoveL 3030 to (53.59, -12.23, 130) mm, rotated rx 180 ry 0 rz 180 deg; joints [27.2, 49.842, 9.151, -149.052, 62.731, -195.362]
  Call Extruder(28481.916)
  MoveL 3031 to (54.97, 0, 130) mm, rotated rx 180 ry 0 rz -180 deg; joints [28.57, 50.879, 7.123, -147.296, 62.266, -196.636]
  Call Extruder(28492.847)
  MoveL 3032 to (53.59, 12.23, 130) mm, rotated rx 180 ry 0 rz -180 deg; joints [30.077, 51.608, 5.699, -145.466, 62.134, -197.83]
  Call Extruder(28503.777)
  MoveL 3033 to (49.53, 23.85, 130) mm, rotated rx 180 ry 0 rz -180 deg; joints [31.665, 51.988, 4.957, -143.651, 62.339, -198.862]
  Call Extruder(28514.707)
  MoveL 3034 to (42.98, 34.27, 130) mm, rotated rx 180 ry 0 rz 180 deg; joints [33.282, 51.999, 4.935, -141.929, 62.864, -199.66]
  Call Extruder(28525.637)
  MoveL 3035 to (34.27, 42.98, 130) mm, rotated rx -180 ry 0 rz 180 deg; joints [34.874, 51.64, 5.636, -140.361, 63.672, -200.174]
  Call Extruder(28536.567)
  MoveL 3036 to (23.85, 49.53, 130) mm, rotated rx 180 ry 0 rz -180 deg; joints [36.387, 50.931, 7.021, -138.996, 64.712, -200.374]
  Call Extruder(28547.498)
  MoveL 3037 to (12.23, 53.59, 130) mm, rotated rx 180 ry 0 rz 180 deg; joints [37.766, 49.911, 9.017, -137.87, 65.921, -200.256]
  Call Extruder(28558.428)
  MoveL 3038 to (0, 54.97, 130) mm, rotated rx 180 ry 0 rz -180 deg; joints [38.954, 48.633, 11.52, -137.012, 67.231, -199.837]
  Call Extruder(28569.358)
  MoveL 3039 to (-12.23, 53.59, 130) mm, rotated rx 180 ry 0 rz -180 deg; joints [39.895, 47.162, 14.407, -136.45, 68.575, -199.149]
  Call Extruder(28580.288)
  MoveL 3040 to (-23.85, 49.52, 130) mm, rotated rx -180 ry 0 rz -180 deg; joints [40.528, 45.568, 17.54, -136.211, 69.892, -198.24]
  Call Extruder(28591.218)
  MoveL 3041 to (-34.27, 42.98, 130) mm, rotated rx 180 ry 0 rz 180 deg; joints [40.799, 43.928, 20.773, -136.327, 71.126, -197.163]
  Call Extruder(28602.149)
  MoveL 3042 to (-42.98, 34.27, 130) mm, rotated rx 180 ry 0 rz -180 deg; joints [40.659, 42.319, 23.954, -136.827, 72.227, -195.98]
  Call Extruder(28613.079)
  MoveL 3043 to (-49.53, 23.85, 130) mm, rotated rx 180 ry 0 rz 180 deg; joints [40.072, 40.818, 26.929, -137.731, 73.155, -194.757]
  Call Extruder(28624.009)
  MoveL 3044 to (-53.59, 12.23, 130) mm, rotated rx -180 ry 0 rz 180 deg; joints [39.031, 39.501, 29.547, -139.04, 73.873, -193.557]
  Call Extruder(28634.939)
  MoveL 3045 to (-54.97, 0, 130) mm, rotated rx 180 ry 0 rz -180 deg; joints [37.56, 38.438, 31.666, -140.723, 74.349, -192.441]
  Call Extruder(28640.465)
  MoveL 3046 to (-54.27, -6.18, 130) mm, rotated rx 180 ry 0 rz 180 deg; joints [36.644, 38.052, 32.436, -141.72, 74.456, -191.941]
  Set speed (130.0 mm/s)
  MoveL 3047 to (-49.9, -9.51, 130) mm, rotated rx 180 ry 0 rz -180 deg; joints [35.741, 38.242, 32.057, -142.605, 74.12, -191.814]
  MoveL 3048 to (2.97, -12.99, 130) mm, rotated rx 180 ry 0 rz 180 deg; joints [30.614, 43.605, 21.411, -146.863, 68.685, -193.349]
  Call Extruder(28645.128)
  Set speed (80.0 mm/s)
  MoveL 3049 to (5.78, -12.01, 130) mm, rotated rx 180 ry 0 rz 180 deg; joints [30.526, 43.993, 20.645, -146.874, 68.348, -193.537]
  Call Extruder(28649.792)
  MoveL 3050 to (8.31, -10.42, 130) mm, rotated rx 180 ry 0 rz -180 deg; joints [30.538, 44.391, 19.859, -146.776, 68.027, -193.771]
  Call Extruder(28654.456)
  MoveL 3051 to (10.42, -8.31, 130) mm, rotated rx 180 ry 0 rz -180 deg; joints [30.649, 44.78, 19.094, -146.576, 67.738, -194.038]
  Call Extruder(28659.120)
  MoveL 3052 to (12.01, -5.78, 130) mm, rotated rx 180 ry 0 rz -180 deg; joints [30.85, 45.139, 18.386, -146.285, 67.497, -194.327]
  Call Extruder(28663.783)
  MoveL 3053 to (12.99, -2.97, 130) mm, rotated rx -180 ry 0 rz 180 deg; joints [31.131, 45.451, 17.771, -145.921, 67.316, -194.623]
  Call Extruder(28668.447)
  MoveL 3054 to (13.33, 0, 130) mm, rotated rx 180 ry 0 rz 180 deg; joints [31.476, 45.701, 17.279, -145.502, 67.204, -194.91]
  Call Extruder(28673.111)
  MoveL 3055 to (12.99, 2.97, 130) mm, rotated rx 180 ry 0 rz 180 deg; joints [31.869, 45.876, 16.935, -145.049, 67.167, -195.174]
  Call Extruder(28677.775)
  MoveL 3056 to (12.01, 5.78, 130) mm, rotated rx -180 ry 0 rz 180 deg; joints [32.292, 45.966, 16.757, -144.586, 67.207, -195.401]
  Call Extruder(28682.439)
  MoveL 3057 to (10.42, 8.31, 130) mm, rotated rx 180 ry 0 rz 180 deg; joints [32.725, 45.969, 16.751, -144.132, 67.32, -195.578]
  Call Extruder(28687.103)
  MoveL 3058 to (8.31, 10.42, 130) mm, rotated rx -180 ry 0 rz -180 deg; joints [33.149, 45.883, 16.92, -143.711, 67.501, -195.694]
  Call Extruder(28691.766)
  MoveL 3059 to (5.78, 12.01, 130) mm, rotated rx -180 ry 0 rz 180 deg; joints [33.544, 45.713, 17.255, -143.339, 67.741, -195.745]
  Call Extruder(28696.430)
  MoveL 3060 to (2.97, 13, 130) mm, rotated rx 180 ry 0 rz -180 deg; joints [33.893, 45.468, 17.738, -143.035, 68.026, -195.728]
  Call Extruder(28701.094)
  MoveL 3061 to (0, 13.33, 130) mm, rotated rx -180 ry 0 rz 180 deg; joints [34.177, 45.159, 18.347, -142.812, 68.342, -195.643]
  Call Extruder(28705.758)
  MoveL 3062 to (-2.97, 13, 130) mm, rotated rx 180 ry 0 rz -180 deg; joints [34.384, 44.802, 19.05, -142.681, 68.673, -195.496]
  Call Extruder(28710.421)
  MoveL 3063 to (-5.78, 12.01, 130) mm, rotated rx 180 ry 0 rz -180 deg; joints [34.5, 44.415, 19.813, -142.65, 69.003, -195.295]
  Call Extruder(28715.085)
  MoveL 3064 to (-8.31, 10.42, 130) mm, rotated rx 180 ry 0 rz 180 deg; joints [34.518, 44.016, 20.599, -142.72, 69.316, -195.05]
  Call Extruder(28719.749)
  MoveL 3065 to (-10.42, 8.31, 130) mm, rotated rx -180 ry 0 rz 180 deg; joints [34.436, 43.627, 21.367, -142.891, 69.597, -194.775]
  Call Extruder(28724.413)
  MoveL 3066 to (-12.01, 5.78, 130) mm, rotated rx 180 ry 0 rz 180 deg; joints [34.254, 43.267, 22.08, -143.156, 69.832, -194.485]
  Call Extruder(28729.076)
  MoveL 3067 to (-12.99, 2.97, 130) mm, rotated rx 180 ry 0 rz -180 deg; joints [33.981, 42.952, 22.701, -143.505, 70.01, -194.193]
  Call Extruder(28733.740)
  MoveL 3068 to (-13.33, 0, 130) mm, rotated rx -180 ry 0 rz -180 deg; joints [33.63, 42.701, 23.198, -143.92, 70.123, -193.915]
  Call Extruder(28738.404)
  MoveL 3069 to (-13, -2.97, 130) mm, rotated rx 180 ry 0 rz -180 deg; joints [33.218, 42.525, 23.547, -144.382, 70.165, -193.663]
  Call Extruder(28743.068)
  MoveL 3070 to (-12.01, -5.78, 130) mm, rotated rx 180 ry 0 rz 180 deg; joints [32.767, 42.433, 23.728, -144.867, 70.132, -193.449]
  Call Extruder(28747.732)
  MoveL 3071 to (-10.42, -8.31, 130) mm, rotated rx -180 ry 0 rz -180 deg; joints [32.302, 42.43, 23.734, -145.348, 70.027, -193.284]
  Call Extruder(28752.396)
  MoveL 3072 to (-8.31, -10.42, 130) mm, rotated rx 180 ry 0 rz 180 deg; joints [31.85, 42.517, 23.562, -145.799, 69.854, -193.174]
  Call Extruder(28757.059)
  MoveL 3073 to (-5.78, -12.01, 130) mm, rotated rx 180 ry 0 rz -180 deg; joints [31.435, 42.688, 23.223, -146.196, 69.62, -193.125]
  Call Extruder(28761.723)
  MoveL 3074 to (-2.97, -12.99, 130) mm, rotated rx -180 ry 0 rz 180 deg; joints [31.079, 42.936, 22.734, -146.515, 69.338, -193.138]
  Call Extruder(28766.387)
  MoveL 3075 to (0, -13.33, 130) mm, rotated rx 180 ry 0 rz -180 deg; joints [30.801, 43.247, 22.119, -146.742, 69.021, -193.214]
  Call Extruder(28771.051)
  MoveL 3076 to (2.97, -12.99, 130) mm, rotated rx 180 ry 0 rz 180 deg; joints [30.614, 43.605, 21.411, -146.863, 68.685, -193.349]
  Set speed (130.0 mm/s)
  MoveL 3077 to (2.97, -12.99, 135) mm, rotated rx 180 ry 0 rz -180 deg; joints [30.614, 42.764, 21.571, -146.715, 68.115, -193.75]
  MoveL 3078 to (-26.25, -4.54, 135) mm, rotated rx -180 ry 0 rz -180 deg; joints [34.172, 40.114, 26.734, -143.559, 71.016, -193.506]
  Call Extruder(28773.283)
  Set speed (60.0 mm/s)
  MoveL 3079 to (-26.09, -5.96, 135) mm, rotated rx 180 ry 0 rz 180 deg; joints [33.969, 40.028, 26.9, -143.785, 71.034, -193.387]
  Call Extruder(28782.648)
  MoveL 3080 to (-24.12, -11.61, 135) mm, rotated rx 180 ry 0 rz 180 deg; joints [33.033, 39.839, 27.27, -144.785, 70.967, -192.962]
  Call Extruder(28792.013)
  MoveL 3081 to (-20.93, -16.69, 135) mm, rotated rx 180 ry 0 rz -180 deg; joints [32.066, 39.833, 27.28, -145.785, 70.757, -192.632]
  Call Extruder(28801.378)
  MoveL 3082 to (-16.69, -20.93, 135) mm, rotated rx 180 ry 0 rz 180 deg; joints [31.126, 40.012, 26.932, -146.724, 70.412, -192.409]
  Call Extruder(28810.743)
  MoveL 3083 to (-11.61, -24.11, 135) mm, rotated rx 180 ry 0 rz 180 deg; joints [30.272, 40.365, 26.243, -147.545, 69.947, -192.301]
  Call Extruder(28820.108)
  MoveL 3084 to (-5.96, -26.09, 135) mm, rotated rx 180 ry 0 rz 180 deg; joints [29.552, 40.874, 25.251, -148.2, 69.385, -192.315]
  Call Extruder(28829.473)
  MoveL 3085 to (0, -26.77, 135) mm, rotated rx -180 ry 0 rz -180 deg; joints [29.003, 41.512, 24.008, -148.653, 68.752, -192.449]
  Call Extruder(28838.838)
  MoveL 3086 to (5.96, -26.09, 135) mm, rotated rx 180 ry 0 rz 180 deg; joints [28.65, 42.246, 22.58, -148.881, 68.081, -192.7]
  Call Extruder(28848.203)
  MoveL 3087 to (11.61, -24.11, 135) mm, rotated rx 180 ry 0 rz 180 deg; joints [28.503, 43.038, 21.038, -148.878, 67.407, -193.059]
  Call Extruder(28857.568)
  MoveL 3088 to (16.69, -20.93, 135) mm, rotated rx 180 ry 0 rz -180 deg; joints [28.559, 43.849, 19.461, -148.65, 66.765, -193.514]
  Call Extruder(28866.933)
  MoveL 3089 to (20.93, -16.69, 135) mm, rotated rx 180 ry 0 rz -180 deg; joints [28.808, 44.64, 17.925, -148.217, 66.189, -194.045]
  Call Extruder(28876.298)
  MoveL 3090 to (24.12, -11.61, 135) mm, rotated rx 180 ry 0 rz -180 deg; joints [29.229, 45.37, 16.506, -147.607, 65.71, -194.627]
  Call Extruder(28885.663)
  MoveL 3091 to (26.09, -5.96, 135) mm, rotated rx 180 ry 0 rz -180 deg; joints [29.796, 46.005, 15.275, -146.857, 65.354, -195.232]
  Call Extruder(28895.028)
  MoveL 3092 to (26.77, 0, 135) mm, rotated rx 180 ry 0 rz -180 deg; joints [30.482, 46.512, 14.29, -146.009, 65.14, -195.826]
  Call Extruder(28904.393)
  MoveL 3093 to (26.09, 5.96, 135) mm, rotated rx 180 ry 0 rz 180 deg; joints [31.252, 46.867, 13.602, -145.105, 65.079, -196.378]
  Call Extruder(28913.758)
  MoveL 3094 to (24.11, 11.61, 135) mm, rotated rx 180 ry 0 rz 180 deg; joints [32.076, 47.052, 13.244, -144.189, 65.173, -196.855]
  Call Extruder(28923.123)
  MoveL 3095 to (20.93, 16.69, 135) mm, rotated rx 180 ry 0 rz 180 deg; joints [32.917, 47.057, 13.233, -143.302, 65.415, -197.228]
  Call Extruder(28932.488)
  MoveL 3096 to (16.69, 20.93, 135) mm, rotated rx 180 ry 0 rz -180 deg; joints [33.742, 46.883, 13.572, -142.482, 65.792, -197.477]
  Call Extruder(28941.853)
  MoveL 3097 to (11.61, 24.12, 135) mm, rotated rx 180 ry 0 rz 180 deg; joints [34.517, 46.537, 14.241, -141.762, 66.282, -197.587]
  Call Extruder(28951.218)
  MoveL 3098 to (5.96, 26.09, 135) mm, rotated rx 180 ry 0 rz -180 deg; joints [35.208, 46.038, 15.21, -141.17, 66.857, -197.554]
  Call Extruder(28960.583)
  MoveL 3099 to (0, 26.77, 135) mm, rotated rx 180 ry 0 rz 180 deg; joints [35.784, 45.41, 16.428, -140.731, 67.489, -197.381]
  Call Extruder(28969.948)
  MoveL 3100 to (-5.96, 26.09, 135) mm, rotated rx 180 ry 0 rz 180 deg; joints [36.214, 44.685, 17.838, -140.465, 68.144, -197.08]
  Call Extruder(28979.313)
  MoveL 3101 to (-11.61, 24.12, 135) mm, rotated rx 180 ry 0 rz -180 deg; joints [36.473, 43.897, 19.368, -140.384, 68.792, -196.669]
  Call Extruder(28988.678)
  MoveL 3102 to (-16.69, 20.93, 135) mm, rotated rx -180 ry 0 rz 180 deg; joints [36.542, 43.086, 20.946, -140.501, 69.402, -196.172]
  Call Extruder(28998.043)
  MoveL 3103 to (-20.93, 16.69, 135) mm, rotated rx 180 ry 0 rz 180 deg; joints [36.407, 42.291, 22.492, -140.816, 69.946, -195.616]
  Call Extruder(29007.408)
  MoveL 3104 to (-24.12, 11.61, 135) mm, rotated rx 180 ry 0 rz -180 deg; joints [36.065, 41.553, 23.929, -141.324, 70.4, -195.03]
  Call Extruder(29016.773)
  MoveL 3105 to (-26.09, 5.96, 135) mm, rotated rx 180 ry 0 rz 180 deg; joints [35.528, 40.909, 25.184, -142.009, 70.742, -194.445]
  Call Extruder(29026.138)
  MoveL 3106 to (-26.77, 0, 135) mm, rotated rx 180 ry 0 rz 180 deg; joints [34.817, 40.391, 26.193, -142.842, 70.958, -193.889]
  Call Extruder(29030.926)
  MoveL 3107 to (-26.42, -3.05, 135) mm, rotated rx 180 ry 0 rz 180 deg; joints [34.385, 40.204, 26.557, -143.323, 70.997, -193.631]
  Set speed (130.0 mm/s)
  MoveL 3108 to (-41.86, -6.29, 135) mm, rotated rx 180 ry 0 rz 180 deg; joints [35.393, 38.352, 30.171, -142.638, 72.635, -192.837]
  Call Extruder(29035.924)
  Set speed (60.0 mm/s)
  MoveL 3109 to (-41.5, -9.47, 135) mm, rotated rx -180 ry 0 rz -180 deg; joints [34.924, 38.159, 30.549, -143.153, 72.679, -192.578]
  Call Extruder(29050.820)
  MoveL 3110 to (-38.36, -18.47, 135) mm, rotated rx 180 ry 0 rz 180 deg; joints [33.373, 37.853, 31.147, -144.794, 72.586, -191.923]
  Call Extruder(29065.716)
  MoveL 3111 to (-33.29, -26.54, 135) mm, rotated rx -180 ry 0 rz -180 deg; joints [31.763, 37.844, 31.165, -146.45, 72.267, -191.419]
  Call Extruder(29080.612)
  MoveL 3112 to (-26.54, -33.28, 135) mm, rotated rx 180 ry 0 rz -180 deg; joints [30.206, 38.133, 30.6, -148.007, 71.731, -191.08]
  Call Extruder(29095.507)
  MoveL 3113 to (-18.47, -38.36, 135) mm, rotated rx 180 ry 0 rz 180 deg; joints [28.808, 38.703, 29.486, -149.361, 71, -190.915]
  Call Extruder(29110.403)
  MoveL 3114 to (-9.47, -41.51, 135) mm, rotated rx -180 ry 0 rz 180 deg; joints [27.654, 39.522, 27.887, -150.424, 70.107, -190.93]
  Call Extruder(29125.299)
  MoveL 3115 to (0, -42.57, 135) mm, rotated rx 180 ry 0 rz 180 deg; joints [26.805, 40.545, 25.893, -151.137, 69.097, -191.126]
  Call Extruder(29140.195)
  MoveL 3116 to (9.47, -41.5, 135) mm, rotated rx -180 ry 0 rz -180 deg; joints [26.29, 41.717, 23.61, -151.469, 68.021, -191.501]
  Call Extruder(29155.091)
  MoveL 3117 to (18.47, -38.36, 135) mm, rotated rx 180 ry 0 rz 180 deg; joints [26.114, 42.979, 21.153, -151.419, 66.936, -192.047]
  Call Extruder(29169.986)
  MoveL 3118 to (26.54, -33.28, 135) mm, rotated rx -180 ry 0 rz -180 deg; joints [26.262, 44.269, 18.646, -151.006, 65.9, -192.75]
  Call Extruder(29184.882)
  MoveL 3119 to (33.28, -26.54, 135) mm, rotated rx -180 ry 0 rz -180 deg; joints [26.703, 45.524, 16.208, -150.268, 64.97, -193.585]
  Call Extruder(29199.778)
  MoveL 3120 to (38.36, -18.47, 135) mm, rotated rx 180 ry 0 rz -180 deg; joints [27.4, 46.684, 13.956, -149.258, 64.197, -194.514]
  Call Extruder(29214.674)
  MoveL 3121 to (41.51, -9.47, 135) mm, rotated rx 180 ry 0 rz 180 deg; joints [28.309, 47.693, 12, -148.04, 63.623, -195.493]
  Call Extruder(29229.570)
  MoveL 3122 to (42.57, 0, 135) mm, rotated rx 180 ry 0 rz 180 deg; joints [29.382, 48.502, 10.434, -146.682, 63.28, -196.466]
  Call Extruder(29244.465)
  MoveL 3123 to (41.5, 9.47, 135) mm, rotated rx 180 ry 0 rz -180 deg; joints [30.575, 49.068, 9.337, -145.254, 63.188, -197.373]
  Call Extruder(29259.361)
  MoveL 3124 to (38.36, 18.47, 135) mm, rotated rx 180 ry 0 rz 180 deg; joints [31.839, 49.363, 8.766, -143.825, 63.348, -198.159]
  Call Extruder(29274.257)
  MoveL 3125 to (33.28, 26.54, 135) mm, rotated rx 180 ry 0 rz -180 deg; joints [33.128, 49.372, 8.749, -142.458, 63.75, -198.773]
  Call Extruder(29289.153)
  MoveL 3126 to (26.54, 33.28, 135) mm, rotated rx -180 ry 0 rz -180 deg; joints [34.394, 49.093, 9.288, -141.204, 64.367, -199.176]
  Call Extruder(29304.049)
  MoveL 3127 to (18.47, 38.36, 135) mm, rotated rx 180 ry 0 rz -180 deg; joints [35.592, 48.542, 10.355, -140.108, 65.161, -199.348]
  Call Extruder(29318.944)
  MoveL 3128 to (9.47, 41.51, 135) mm, rotated rx 180 ry 0 rz -180 deg; joints [36.675, 47.747, 11.896, -139.205, 66.087, -199.281]
  Call Extruder(29333.840)
  MoveL 3129 to (0, 42.57, 135) mm, rotated rx 180 ry 0 rz -180 deg; joints [37.594, 46.748, 13.832, -138.526, 67.095, -198.985]
  Call Extruder(29348.736)
  MoveL 3130 to (-9.47, 41.51, 135) mm, rotated rx 180 ry 0 rz -180 deg; joints [38.304, 45.595, 16.069, -138.095, 68.133, -198.482]
  Call Extruder(29363.632)
  MoveL 3131 to (-18.47, 38.36, 135) mm, rotated rx 180 ry 0 rz -180 deg; joints [38.762, 44.344, 18.499, -137.936, 69.152, -197.805]
  Call Extruder(29378.528)
  MoveL 3132 to (-26.54, 33.28, 135) mm, rotated rx -180 ry 0 rz -180 deg; joints [38.928, 43.055, 21.006, -138.07, 70.106, -196.995]
  Call Extruder(29393.423)
  MoveL 3133 to (-33.29, 26.54, 135) mm, rotated rx 180 ry 0 rz -180 deg; joints [38.772, 41.789, 23.469, -138.51, 70.955, -196.098]
  Call Extruder(29408.319)
  MoveL 3134 to (-38.36, 18.47, 135) mm, rotated rx 180 ry 0 rz -180 deg; joints [38.277, 40.61, 25.766, -139.262, 71.664, -195.16]
  Call Extruder(29423.215)
  MoveL 3135 to (-41.51, 9.47, 135) mm, rotated rx 180 ry 0 rz 180 deg; joints [37.447, 39.577, 27.78, -140.314, 72.203, -194.232]
  Call Extruder(29438.111)
  MoveL 3136 to (-42.57, 0, 135) mm, rotated rx -180 ry 0 rz -180 deg; joints [36.31, 38.745, 29.404, -141.63, 72.547, -193.358]
  Call Extruder(29445.665)
  MoveL 3137 to (-42.03, -4.8, 135) mm, rotated rx 180 ry 0 rz 180 deg; joints [35.612, 38.444, 29.992, -142.398, 72.614, -192.959]
  Set speed (130.0 mm/s)
  MoveL 3138 to (-54.1, -7.67, 135) mm, rotated rx 180 ry 0 rz 180 deg; joints [36.421, 37.015, 32.786, -141.826, 73.868, -192.322]
  Call Extruder(29449.738)
  Set speed (30.0 mm/s)
  MoveL 3139 to (-53.59, -12.23, 135) mm, rotated rx 180 ry 0 rz -180 deg; joints [35.732, 36.735, 33.333, -142.575, 73.935, -191.957]
  Call Extruder(29460.668)
  MoveL 3140 to (-49.53, -23.85, 135) mm, rotated rx -180 ry 0 rz -180 deg; joints [33.663, 36.333, 34.12, -144.751, 73.831, -191.134]
  Call Extruder(29471.598)
  MoveL 3141 to (-42.98, -34.27, 135) mm, rotated rx 180 ry 0 rz 180 deg; joints [31.506, 36.322, 34.143, -146.961, 73.435, -190.505]
  Call Extruder(29482.528)
  MoveL 3142 to (-34.27, -42.98, 135) mm, rotated rx -180 ry 0 rz -180 deg; joints [29.427, 36.701, 33.4, -149.04, 72.755, -190.084]
  Call Extruder(29493.458)
  MoveL 3143 to (-23.85, -49.53, 135) mm, rotated rx -180 ry 0 rz 180 deg; joints [27.581, 37.447, 31.94, -150.835, 71.818, -189.879]
  Call Extruder(29504.389)
  MoveL 3144 to (-12.23, -53.59, 135) mm, rotated rx -180 ry 0 rz -180 deg; joints [26.087, 38.516, 29.852, -152.224, 70.665, -189.892]
  Call Extruder(29515.319)
  MoveL 3145 to (0, -54.97, 135) mm, rotated rx 180 ry 0 rz 180 deg; joints [25.019, 39.845, 27.257, -153.132, 69.355, -190.128]
  Call Extruder(29524.699)
  MoveL 3146 to (10.5, -53.79, 135) mm, rotated rx 180 ry 0 rz -180 deg; joints [24.49, 41.146, 24.722, -153.474, 68.157, -190.521]
  Call Extruder(29526.249)
  MoveL 3147 to (12.23, -53.59, 135) mm, rotated rx 180 ry 0 rz -180 deg; joints [24.406, 41.364, 24.297, -153.527, 67.957, -190.587]
  Call Extruder(29537.179)
  MoveL 3148 to (23.85, -49.52, 135) mm, rotated rx -180 ry 0 rz -180 deg; joints [24.239, 42.994, 21.123, -153.415, 66.544, -191.266]
  Call Extruder(29548.109)
  MoveL 3149 to (34.27, -42.98, 135) mm, rotated rx 180 ry 0 rz -180 deg; joints [24.487, 44.659, 17.888, -152.83, 65.193, -192.153]
  Call Extruder(29559.040)
  MoveL 3150 to (42.98, -34.27, 135) mm, rotated rx 180 ry 0 rz 180 deg; joints [25.101, 46.278, 14.744, -151.831, 63.978, -193.221]
  Call Extruder(29569.970)
  MoveL 3151 to (49.52, -23.85, 135) mm, rotated rx 180 ry 0 rz -180 deg; joints [26.025, 47.777, 11.838, -150.489, 62.966, -194.427]
  Call Extruder(29580.900)
  MoveL 3152 to (53.59, -12.23, 135) mm, rotated rx 180 ry 0 rz 180 deg; joints [27.2, 49.082, 9.31, -148.89, 62.215, -195.712]
  Call Extruder(29591.830)
  MoveL 3153 to (54.97, 0, 135) mm, rotated rx 180 ry 0 rz 180 deg; joints [28.57, 50.13, 7.282, -147.126, 61.769, -196.999]
  Call Extruder(29602.760)
  MoveL 3154 to (53.59, 12.23, 135) mm, rotated rx 180 ry 0 rz -180 deg; joints [30.077, 50.865, 5.859, -145.289, 61.654, -198.206]
  Call Extruder(29613.691)
  MoveL 3155 to (49.52, 23.85, 135) mm, rotated rx 180 ry 0 rz 180 deg; joints [31.665, 51.249, 5.116, -143.469, 61.872, -199.251]
  Call Extruder(29624.621)
  MoveL 3156 to (42.98, 34.27, 135) mm, rotated rx 180 ry 0 rz 180 deg; joints [33.282, 51.26, 5.095, -141.744, 62.408, -200.063]
  Call Extruder(29635.551)
  MoveL 3157 to (34.27, 42.98, 135) mm, rotated rx 180 ry 0 rz 180 deg; joints [34.874, 50.898, 5.796, -140.175, 63.224, -200.59]
  Call Extruder(29646.481)
